KUKA KRL program: MyProgram_274().src

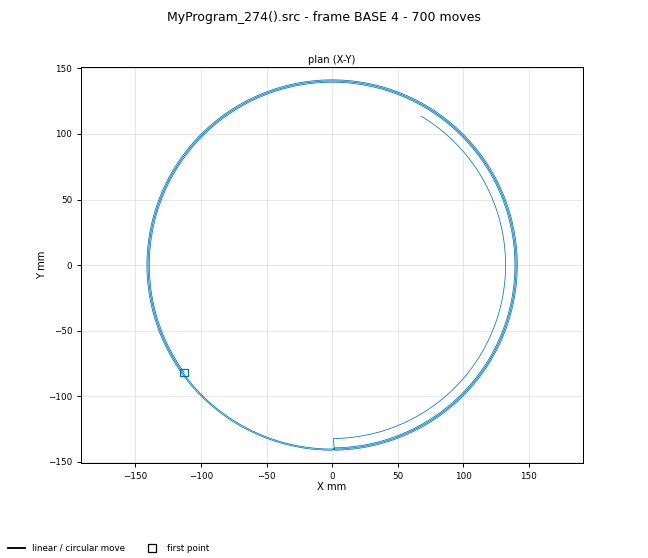
[picture p0: tool path of MyProgram_274().src in frame BASE 4, 700 of 700 moves have a stored position in this frame; points joined in program order, loops and branches not executed]
&ACCESS RVP
&REL 1
&PARAM TEMPLATE = C:\KRC\Roboter\Template\vorgabe
&PARAM EDITMASK = *
DEF MyProgram_274()
; ---- Setting reference (Base) ----
$BASE = BASE_DATA[4]

; --------------------------
; ---- Setting tool (TCP) ----
$TOOL = TOOL_DATA[3]
; --------------------------

$VEL.CP = VEL_APROX_PRINT
Startdeposition()
$VEL.CP = VEL_PRINT
LIN {X -112.8396,Y -81.9859,Z 171,A -142.2331,B 8.8363,C 0.3441,E1 8.7131,E2 233.8465} C_DIS
LIN {X -115.5145,Y -78.1719,Z 171,A -144.1484,B 8.8365,C 0.3397,E1 8.71,E2 235.7611} C_DIS
LIN {X -118.0573,Y -74.2762,Z 171,A -146.0937,B 8.8366,C 0.3357,E1 8.7071,E2 237.7098} C_DIS
LIN {X -120.4012,Y -70.4136,Z 171,A -147.8161,B 8.8369,C 0.3289,E1 8.7047,E2 239.4141} C_DIS
LIN {X -122.1598,Y -67.3164,Z 171,A -149.6524,B 8.8368,C 0.3315,E1 8.7021,E2 241.297} C_DIS
LIN {X -124.439,Y -62.9993,Z 171,A -151.4139,B 8.8371,C 0.3224,E1 8.6999,E2 243.0262} C_DIS
LIN {X -125.9748,Y -59.8691,Z 171,A -152.8774,B 8.8372,C 0.3192,E1 8.6981,E2 244.4928} C_DIS
LIN {X -127.4555,Y -56.6489,Z 171,A -154.3628,B 8.8374,C 0.3159,E1 8.6964,E2 245.981} C_DIS
LIN {X -128.9714,Y -53.1107,Z 171,A -156.2039,B 8.8374,C 0.3161,E1 8.6944,E2 247.854} C_DIS
LIN {X -130.384,Y -49.5416,Z 171,A -158.0959,B 8.8374,C 0.3171,E1 8.6925,E2 249.7847} C_DIS
LIN {X -131.9696,Y -45.1472,Z 171,A -159.478,B 8.8378,C 0.303,E1 8.6913,E2 251.0977} C_DIS
LIN {X -132.9491,Y -42.1728,Z 171,A -160.7834,B 8.8379,C 0.2998,E1 8.6901,E2 252.4044} C_DIS
LIN {X -133.9563,Y -38.8556,Z 171,A -162.2355,B 8.838,C 0.2964,E1 8.689,E2 253.8591} C_DIS
LIN {X -134.8227,Y -35.7326,Z 171,A -163.6103,B 8.8381,C 0.2934,E1 8.688,E2 255.2384} C_DIS
LIN {X -135.806,Y -31.8005,Z 171,A -165.4341,B 8.8382,C 0.2913,E1 8.6867,E2 257.081} C_DIS
LIN {X -136.6688,Y -27.8498,Z 171,A -167.0113,B 8.8384,C 0.2853,E1 8.6858,E2 258.6461} C_DIS
LIN {X -137.3745,Y -24.1335,Z 171,A -168.6614,B 8.8384,C 0.2824,E1 8.685,E2 260.3072} C_DIS
LIN {X -138.0563,Y -19.8611,Z 171,A -170.4155,B 8.8387,C 0.277,E1 8.6843,E2 262.0568} C_DIS
LIN {X -138.5691,Y -15.906,Z 171,A -172.5929,B 8.8385,C 0.281,E1 8.6836,E2 264.3005} C_DIS
LIN {X -139.0257,Y -11.2308,Z 171,A -173.9284,B 8.839,C 0.2658,E1 8.6833,E2 265.5598} C_DIS
LIN {X -139.2374,Y -8.1929,Z 171,A -175.9129,B 8.8387,C 0.2741,E1 8.6829,E2 267.6352} C_DIS
LIN {X -139.4478,Y -2.9637,Z 171,A -178.1689,B 8.8389,C 0.2696,E1 8.6828,E2 269.9025} C_DIS
LIN {X -139.4551,Y 2.5197,Z 171,A -179.7814,B 8.8394,C 0.2527,E1 8.6828,E2 271.4329} C_DIS
LIN {X -139.0897,Y 10.3992,Z 171,A 177.172,B 8.8397,C 0.2402,E1 8.6833,E2 274.4521} C_DIS
LIN {X -138.4769,Y 16.6784,Z 171,A 174.2904,B 8.8398,C 0.2375,E1 8.6841,E2 277.3677} C_DIS
LIN {X -137.9353,Y 20.6949,Z 171,A 172.3629,B 8.8398,C 0.2369,E1 8.6848,E2 279.3266} C_DIS
LIN {X -137.0859,Y 25.7227,Z 171,A 170.4087,B 8.84,C 0.2286,E1 8.6858,E2 281.2611} C_DIS
LIN {X -136.3153,Y 29.5315,Z 171,A 168.8667,B 8.8402,C 0.2232,E1 8.6867,E2 282.7947} C_DIS
LIN {X -135.543,Y 32.8954,Z 171,A 167.4503,B 8.8402,C 0.2192,E1 8.6876,E2 284.2094} C_DIS
LIN {X -134.7496,Y 36.0069,Z 171,A 166.0979,B 8.8403,C 0.216,E1 8.6885,E2 285.5647} C_DIS
LIN {X -133.815,Y 39.3382,Z 171,A 164.6154,B 8.8404,C 0.213,E1 8.6897,E2 287.0534} C_DIS
LIN {X -132.7678,Y 42.7402,Z 171,A 163.1696,B 8.8405,C 0.2087,E1 8.6909,E2 288.4957} C_DIS
LIN {X -131.6755,Y 45.9954,Z 171,A 161.7245,B 8.8405,C 0.2053,E1 8.6922,E2 289.9437} C_DIS
LIN {X -130.5628,Y 49.0642,Z 171,A 160.3436,B 8.8407,C 0.2023,E1 8.6935,E2 291.3282} C_DIS
LIN {X -129.2438,Y 52.4408,Z 171,A 158.8394,B 8.8407,C 0.1985,E1 8.6951,E2 292.8328} C_DIS
LIN {X -127.8789,Y 55.6868,Z 171,A 157.399,B 8.8408,C 0.1946,E1 8.6967,E2 294.2709} C_DIS
LIN {X -126.442,Y 58.8765,Z 171,A 155.9105,B 8.8409,C 0.1916,E1 8.6984,E2 295.7643} C_DIS
LIN {X -124.8829,Y 62.1157,Z 171,A 154.4187,B 8.8409,C 0.188,E1 8.7002,E2 297.2566} C_DIS
LIN {X -123.3331,Y 65.1378,Z 171,A 153.0073,B 8.8411,C 0.1846,E1 8.7021,E2 298.6685} C_DIS
LIN {X -121.1822,Y 69.0604,Z 171,A 150.9956,B 8.8411,C 0.1828,E1 8.7048,E2 300.7001} C_DIS
LIN {X -118.3623,Y 73.7886,Z 171,A 148.7116,B 8.8411,C 0.1775,E1 8.7081,E2 302.9845} C_DIS
LIN {X -116.2771,Y 77.034,Z 171,A 147.1234,B 8.8413,C 0.1737,E1 8.7106,E2 304.5716} C_DIS
LIN {X -113.7268,Y 80.7516,Z 171,A 145.2756,B 8.8413,C 0.1692,E1 8.7135,E2 306.417} C_DIS
LIN {X -111.0828,Y 84.3518,Z 171,A 143.2119,B 8.8413,C 0.1687,E1 8.717,E2 308.5072} C_DIS
LIN {X -109.099,Y 86.9014,Z 171,A 142.3013,B 8.8416,C 0.1587,E1 8.7185,E2 309.3647} C_DIS
LIN {X -107.0989,Y 89.3555,Z 171,A 140.6991,B 8.8416,C 0.1608,E1 8.7214,E2 311.0032} C_DIS
LIN {X -103.7086,Y 93.2685,Z 171,A 138.204,B 8.8415,C 0.1623,E1 8.7261,E2 313.5417} C_DIS
LIN {X -100.7826,Y 96.4226,Z 171,A 137.0283,B 8.8417,C 0.1486,E1 8.7282,E2 314.6424} C_DIS
LIN {X -98.5108,Y 98.7428,Z 171,A 134.866,B 8.8415,C 0.1598,E1 8.7327,E2 316.9059} C_DIS
LIN {X -94.6241,Y 102.4735,Z 171,A 132.7583,B 8.8416,C 0.1536,E1 8.737,E2 318.9986} C_DIS
LIN {X -91.1481,Y 105.5769,Z 171,A 131.3887,B 8.8419,C 0.1406,E1 8.7397,E2 320.299} C_DIS
LIN {X -88.0504,Y 108.1742,Z 171,A 129.1579,B 8.8417,C 0.1473,E1 8.7447,E2 322.5987} C_DIS
LIN {X -84.45,Y 111.0073,Z 171,A 127.7852,B 8.8419,C 0.1352,E1 8.7476,E2 323.9068} C_DIS
LIN {X -81.9039,Y 112.899,Z 171,A 126.4687,B 8.8419,C 0.1332,E1 8.7505,E2 325.2238} C_DIS
LIN {X -78.5911,Y 115.2304,Z 171,A 124.6683,B 8.8419,C 0.1327,E1 8.7547,E2 327.0397} C_DIS
LIN {X -73.9341,Y 118.2721,Z 171,A 122.4186,B 8.842,C 0.1285,E1 8.76,E2 329.283} C_DIS
LIN {X -67.4741,Y 122.0725,Z 171,A 119.5001,B 8.8421,C 0.1211,E1 8.767,E2 332.179} C_DIS
LIN {X -64.5541,Y 123.6396,Z 171,A 117.9816,B 8.8421,C 0.122,E1 8.7708,E2 333.7158} C_DIS
LIN {X -60.8845,Y 125.4897,Z 171,A 116.0518,B 8.8421,C 0.1241,E1 8.7757,E2 335.6743} C_DIS
LIN {X -56.6171,Y 127.4697,Z 171,A 114.3186,B 8.8421,C 0.1182,E1 8.78,E2 337.3812} C_DIS
LIN {X -51.3124,Y 129.6975,Z 171,A 112.0212,B 8.8422,C 0.1144,E1 8.7859,E2 339.6686} C_DIS
LIN {X -46.4257,Y 131.5259,Z 171,A 109.7822,B 8.8422,C 0.1139,E1 8.7918,E2 341.918} C_DIS
LIN {X -42.2053,Y 132.9387,Z 171,A 108.0067,B 8.8422,C 0.1113,E1 8.7965,E2 343.6856} C_DIS
LIN {X -39.0862,Y 133.8888,Z 171,A 106.6832,B 8.8422,C 0.1098,E1 8.8,E2 345.0061} C_DIS
LIN {X -35.8913,Y 134.7804,Z 171,A 105.2586,B 8.8422,C 0.1098,E1 8.8039,E2 346.4375} C_DIS
LIN {X -32.6408,Y 135.6043,Z 171,A 103.8694,B 8.8422,C 0.1091,E1 8.8077,E2 347.8272} C_DIS
LIN {X -28.9193,Y 136.4475,Z 171,A 101.9482,B 8.8422,C 0.1146,E1 8.813,E2 349.7913} C_DIS
LIN {X -25.2244,Y 137.1792,Z 171,A 99.9513,B 8.8422,C 0.1221,E1 8.8187,E2 351.8423} C_DIS
LIN {X -19.1774,Y 138.154,Z 171,A 98.2705,B 8.8423,C 0.1055,E1 8.823,E2 353.4189} C_DIS
LIN {X -15.6692,Y 138.5966,Z 171,A 96.225,B 8.8423,C 0.1161,E1 8.8289,E2 355.5369} C_DIS
LIN {X -10.9093,Y 139.0524,Z 171,A 94.6783,B 8.8423,C 0.1077,E1 8.8331,E2 357.0311} C_DIS
LIN {X -5.1132,Y 139.3843,Z 171,A 92.579,B 8.8423,C 0.1019,E1 8.8388,E2 359.0936} C_DIS
LIN {X -2.0688,Y 139.4626,Z 171,A 91.1654,B 8.8423,C 0.1049,E1 8.8428,E2 360.5269} C_DIS
LIN {X 1.9636,Y 139.4644,Z 171,A 89.1838,B 8.8423,C 0.1111,E1 8.8484,E2 362.548} C_DIS
LIN {X 5.4905,Y 139.3696,Z 171,A 87.8031,B 8.8423,C 0.1099,E1 8.8523,E2 363.9196} C_DIS
LIN {X 9.6693,Y 139.143,Z 171,A 86.2944,B 8.8423,C 0.1062,E1 8.8564,E2 365.4017} C_DIS
LIN {X 13.7603,Y 138.7979,Z 171,A 84.3806,B 8.8423,C 0.111,E1 8.8618,E2 367.343} C_DIS
LIN {X 17.0865,Y 138.4282,Z 171,A 83.2481,B 8.8423,C 0.1067,E1 8.8649,E2 368.4449} C_DIS
LIN {X 23.7404,Y 137.4444,Z 171,A 80.562,B 8.8423,C 0.1064,E1 8.8723,E2 371.1207} C_DIS
LIN {X 32.9569,Y 135.5281,Z 171,A 76.6599,B 8.8423,C 0.1094,E1 8.8829,E2 375.0263} C_DIS
LIN {X 36.1847,Y 134.7022,Z 171,A 75.3275,B 8.8423,C 0.1096,E1 8.8865,E2 376.3539} C_DIS
LIN {X 39.3671,Y 133.8066,Z 171,A 73.9683,B 8.8423,C 0.1107,E1 8.8901,E2 377.713} C_DIS
LIN {X 42.5681,Y 132.8228,Z 171,A 72.5899,B 8.8423,C 0.1119,E1 8.8938,E2 379.0915} C_DIS
LIN {X 46.0136,Y 131.6692,Z 171,A 71.1204,B 8.8423,C 0.1128,E1 8.8977,E2 380.558} C_DIS
LIN {X 49.2886,Y 130.4787,Z 171,A 69.7052,B 8.8423,C 0.1139,E1 8.9014,E2 381.971} C_DIS
LIN {X 52.7987,Y 129.0996,Z 171,A 67.8474,B 8.8421,C 0.1219,E1 8.9063,E2 383.8671} C_DIS
LIN {X 55.9083,Y 127.7831,Z 171,A 66.7646,B 8.8421,C 0.1172,E1 8.909,E2 384.9119} C_DIS
LIN {X 61.6274,Y 125.1238,Z 171,A 63.7194,B 8.8421,C 0.1297,E1 8.9168,E2 388.0136} C_DIS
LIN {X 65.6766,Y 123.0495,Z 171,A 62.2846,B 8.8421,C 0.1233,E1 8.9202,E2 389.3945} C_DIS
LIN {X 69.451,Y 120.9593,Z 171,A 60.5123,B 8.8421,C 0.1257,E1 8.9245,E2 391.1669} C_DIS
LIN {X 73.3803,Y 118.6167,Z 171,A 58.8119,B 8.8421,C 0.1248,E1 8.9285,E2 392.8451} C_DIS
LIN {X 75.557,Y 117.2423,Z 171,A 57.3892,B 8.842,C 0.1341,E1 8.932,E2 394.3136} C_DIS
LIN {X 78.2884,Y 115.4356,Z 171,A 55.6399,B 8.8418,C 0.1446,E1 8.9361,E2 396.1132} C_DIS
LIN {X 82.9019,Y 112.169,Z 171,A 54.0025,B 8.842,C 0.1342,E1 8.9396,E2 397.6659} C_DIS
LIN {X 86.2917,Y 109.5819,Z 171,A 52.2349,B 8.842,C 0.1376,E1 8.9435,E2 399.4358} C_DIS
LIN {X 89.8009,Y 106.7252,Z 171,A 50.3797,B 8.8419,C 0.1409,E1 8.9475,E2 401.2909} C_DIS
LIN {X 93.2101,Y 103.761,Z 171,A 48.3871,B 8.8417,C 0.1473,E1 8.9517,E2 403.3013} C_DIS
LIN {X 96.2147,Y 100.9812,Z 171,A 46.8805,B 8.8417,C 0.1469,E1 8.9548,E2 404.7864} C_DIS
LIN {X 99.2554,Y 97.9949,Z 171,A 45.119,B 8.8417,C 0.1507,E1 8.9582,E2 406.5499} C_DIS
LIN {X 104.0961,Y 92.8361,Z 171,A 42.2829,B 8.8417,C 0.1553,E1 8.9636,E2 409.3782} C_DIS
LIN {X 107.0425,Y 89.4227,Z 171,A 40.4474,B 8.8415,C 0.159,E1 8.9669,E2 411.2124} C_DIS
LIN {X 109.9181,Y 85.8638,Z 171,A 38.6101,B 8.8415,C 0.1623,E1 8.9701,E2 413.0452} C_DIS
LIN {X 112.6381,Y 82.2633,Z 171,A 36.7415,B 8.8415,C 0.1669,E1 8.9732,E2 414.9166} C_DIS
LIN {X 115.3005,Y 78.488,Z 171,A 34.8656,B 8.8413,C 0.1709,E1 8.9762,E2 416.7906} C_DIS
LIN {X 117.4671,Y 75.2058,Z 171,A 33.1544,B 8.8413,C 0.1769,E1 8.9788,E2 418.5148} C_DIS
LIN {X 120.6812,Y 69.932,Z 171,A 30.8465,B 8.8412,C 0.1781,E1 8.9821,E2 420.7952} C_DIS
LIN {X 122.717,Y 66.2955,Z 171,A 29.0961,B 8.8411,C 0.1833,E1 8.9845,E2 422.5514} C_DIS
LIN {X 124.4992,Y 62.8809,Z 171,A 27.6221,B 8.8411,C 0.1849,E1 8.9863,E2 424.0126} C_DIS
LIN {X 126.3601,Y 59.0537,Z 171,A 26.0265,B 8.8411,C 0.186,E1 8.9882,E2 425.5901} C_DIS
LIN {X 129.537,Y 51.7135,Z 171,A 22.7043,B 8.8408,C 0.1956,E1 8.9919,E2 428.9191} C_DIS
LIN {X 130.6783,Y 48.7557,Z 171,A 21.3935,B 8.8408,C 0.1993,E1 8.9932,E2 430.2319} C_DIS
LIN {X 131.9118,Y 45.3138,Z 171,A 19.9147,B 8.8407,C 0.2028,E1 8.9945,E2 431.7089} C_DIS
LIN {X 132.9524,Y 42.1625,Z 171,A 18.5801,B 8.8406,C 0.2059,E1 8.9957,E2 433.0408} C_DIS
LIN {X 133.9281,Y 38.9519,Z 171,A 17.2266,B 8.8406,C 0.2092,E1 8.9968,E2 434.3922} C_DIS
LIN {X 134.8223,Y 35.7344,Z 171,A 15.8718,B 8.8404,C 0.2126,E1 8.9978,E2 435.7459} C_DIS
LIN {X 135.7933,Y 31.8549,Z 171,A 13.7509,B 8.84,C 0.228,E1 8.9992,E2 437.9288} C_DIS
LIN {X 136.7354,Y 27.5224,Z 171,A 12.4936,B 8.8402,C 0.2204,E1 8.9999,E2 439.116} C_DIS
LIN {X 137.2961,Y 24.5712,Z 171,A 10.5895,B 8.8398,C 0.2391,E1 9.0008,E2 441.1061} C_DIS
LIN {X 138.1564,Y 19.161,Z 171,A 9.0747,B 8.84,C 0.2289,E1 9.0014,E2 442.5296} C_DIS
LIN {X 138.8069,Y 13.666,Z 171,A 6.988,B 8.84,C 0.2312,E1 9.0021,E2 444.5945} C_DIS
LIN {X 139.0649,Y 10.7379,Z 171,A 5.5151,B 8.8397,C 0.2407,E1 9.0024,E2 446.1024} C_DIS
LIN {X 139.3175,Y 6.6909,Z 171,A 3.7156,B 8.8395,C 0.2486,E1 9.0027,E2 447.9204} C_DIS
LIN {X 139.482,Y -0.0033,Z 171,A 1.0113,B 8.8393,C 0.2555,E1 9.0027,E2 450.6215} C_DIS
LIN {X 139.398,Y -4.764,Z 171,A -1.0684,B 8.8391,C 0.264,E1 9.0026,E2 452.7187} C_DIS
LIN {X 139.2074,Y -8.6797,Z 171,A -2.2767,B 8.8391,C 0.2596,E1 9.0024,E2 453.8771} C_DIS
LIN {X 138.7329,Y -14.4036,Z 171,A -4.4383,B 8.8391,C 0.2619,E1 9.0019,E2 456.0157} C_DIS
LIN {X 138.2511,Y -18.4595,Z 171,A -6.2004,B 8.8389,C 0.2687,E1 9.0013,E2 457.7903} C_DIS
LIN {X 137.7385,Y -21.9657,Z 171,A -7.7867,B 8.8387,C 0.2758,E1 9.0006,E2 459.3948} C_DIS
LIN {X 137.1068,Y -25.6126,Z 171,A -9.5205,B 8.8384,C 0.285,E1 8.9997,E2 461.1574} C_DIS
LIN {X 136.3613,Y -29.3186,Z 171,A -10.3994,B 8.8387,C 0.2741,E1 8.9993,E2 461.9514} C_DIS
LIN {X 134.8966,Y -35.4555,Z 171,A -13.0858,B 8.8385,C 0.2837,E1 8.9975,E2 464.6527} C_DIS
LIN {X 133.7501,Y -39.5598,Z 171,A -14.9247,B 8.8382,C 0.2906,E1 8.9961,E2 466.5048} C_DIS
LIN {X 132.7916,Y -42.6657,Z 171,A -16.2571,B 8.8382,C 0.2943,E1 8.9949,E2 467.8381} C_DIS
LIN {X 131.6179,Y -46.1617,Z 171,A -17.7427,B 8.838,C 0.2978,E1 8.9936,E2 469.3216} C_DIS
LIN {X 129.7219,Y -51.2517,Z 171,A -19.9243,B 8.8378,C 0.3028,E1 8.9915,E2 471.4991} C_DIS
LIN {X 128.6777,Y -53.8139,Z 171,A -21.0297,B 8.8378,C 0.3052,E1 8.9903,E2 472.6017} C_DIS
LIN {X 125.5512,Y -60.7557,Z 171,A -23.9014,B 8.8376,C 0.3078,E1 8.987,E2 475.4437} C_DIS
LIN {X 123.9373,Y -63.9846,Z 171,A -25.5965,B 8.8373,C 0.3165,E1 8.9848,E2 477.1679} C_DIS
LIN {X 121.4883,Y -68.5207,Z 171,A -27.7719,B 8.8371,C 0.3233,E1 8.9819,E2 479.3529} C_DIS
LIN {X 119.1489,Y -72.513,Z 171,A -29.8109,B 8.8368,C 0.3313,E1 8.9789,E2 481.4117} C_DIS
LIN {X 116.1482,Y -77.2275,Z 171,A -31.9345,B 8.8368,C 0.3331,E1 8.9757,E2 483.5155} C_DIS
LIN {X 112.7181,Y -82.1535,Z 171,A -34.1008,B 8.8368,C 0.3324,E1 8.9723,E2 485.6457} C_DIS
LIN {X 108.5305,Y -87.6104,Z 171,A -37.0675,B 8.8364,C 0.3422,E1 8.9672,E2 488.6336} C_DIS
LIN {X 105.9236,Y -90.7456,Z 171,A -38.816,B 8.8362,C 0.3477,E1 8.964,E2 490.3934} C_DIS
LIN {X 102.2707,Y -94.8428,Z 171,A -41.2535,B 8.8358,C 0.3567,E1 8.9594,E2 492.8566} C_DIS
LIN {X 99.7954,Y -97.4444,Z 171,A -42.5038,B 8.8358,C 0.355,E1 8.957,E2 494.0795} C_DIS
LIN {X 96.4987,Y -100.7098,Z 171,A -44.3704,B 8.8358,C 0.3581,E1 8.9533,E2 495.9428} C_DIS
LIN {X 92.2815,Y -104.5877,Z 171,A -46.9905,B 8.8353,C 0.3687,E1 8.9478,E2 498.5996} C_DIS
LIN {X 89.2531,Y -107.1842,Z 171,A -48.3219,B 8.8355,C 0.3652,E1 8.945,E2 499.8929} C_DIS
LIN {X 85.6888,Y -110.0543,Z 171,A -50.1537,B 8.8354,C 0.3677,E1 8.941,E2 501.7203} C_DIS
LIN {X 82.0331,Y -112.8054,Z 171,A -51.9295,B 8.8354,C 0.3688,E1 8.9371,E2 503.4844} C_DIS
LIN {X 77.9243,Y -115.6821,Z 171,A -53.9797,B 8.8352,C 0.3722,E1 8.9323,E2 505.5352} C_DIS
LIN {X 73.1326,Y -118.7684,Z 171,A -56.5354,B 8.8348,C 0.3807,E1 8.9262,E2 508.1208} C_DIS
LIN {X 69.1462,Y -121.1332,Z 171,A -58.0542,B 8.8351,C 0.3754,E1 8.9227,E2 509.5913} C_DIS
LIN {X 66.3121,Y -122.708,Z 171,A -59.6043,B 8.8348,C 0.3821,E1 8.9188,E2 511.1709} C_DIS
LIN {X 62.9686,Y -124.4546,Z 171,A -61.0442,B 8.8348,C 0.3819,E1 8.9153,E2 512.5978} C_DIS
LIN {X 59.6859,Y -126.0623,Z 171,A -62.6688,B 8.8346,C 0.3866,E1 8.9111,E2 514.2396} C_DIS
LIN {X 53.7609,Y -128.6999,Z 171,A -64.8604,B 8.8349,C 0.38,E1 8.9057,E2 516.372} C_DIS
LIN {X 49.776,Y -130.2955,Z 171,A -67.0581,B 8.8344,C 0.3912,E1 8.8998,E2 518.6276} C_DIS
LIN {X 42.2179,Y -132.9347,Z 171,A -70.1748,B 8.8344,C 0.3911,E1 8.8917,E2 521.7245} C_DIS
LIN {X 38.9371,Y -133.9325,Z 171,A -71.5708,B 8.8344,C 0.3921,E1 8.8879,E2 523.1199} C_DIS
LIN {X 35.5501,Y -134.8714,Z 171,A -73.8381,B 8.8335,C 0.4104,E1 8.8815,E2 525.4944} C_DIS
LIN {X 29.5341,Y -136.3147,Z 171,A -76.3675,B 8.8335,C 0.412,E1 8.8746,E2 528.0238} C_DIS
LIN {X 23.4129,Y -137.4992,Z 171,A -78.2991,B 8.8339,C 0.4008,E1 8.8695,E2 529.8761} C_DIS
LIN {X 17.17,Y -138.4183,Z 171,A -80.6166,B 8.8341,C 0.3966,E1 8.8632,E2 532.1597} C_DIS
LIN {X 14.6108,Y -138.7106,Z 171,A -81.7114,B 8.8341,C 0.3978,E1 8.8601,E2 533.2598} C_DIS
LIN {X 10.9284,Y -139.0508,Z 171,A -83.4594,B 8.8339,C 0.403,E1 8.8552,E2 535.0383} C_DIS
LIN {X 6.5695,Y -139.3236,Z 171,A -85.1821,B 8.8339,C 0.402,E1 8.8504,E2 536.7527} C_DIS
LIN {X 2.1826,Y -139.4608,Z 171,A -86.8306,B 8.834,C 0.3993,E1 8.8459,E2 538.382} C_DIS
LIN {X 2.1826,Y -139.4608,Z 171,A -86.8306,B 8.834,C 0.3993,E1 8.8459,E2 538.382} C_DIS
Enddeposition()
LIN {X 1.0238,Y -140.3815,Z 171,A -86.8855,B 8.834,C 0.3961,E1 8.8457,E2 538.416} C_DIS
Startdeposition()
$VEL.CP = VEL_PRINT
LIN {X 4.1318,Y -140.3274,Z 171,A -85.3306,B 8.8343,C 0.39,E1 8.8501,E2 536.8229} C_DIS
LIN {X 8.0102,Y -140.1607,Z 171,A -83.7344,B 8.8343,C 0.3893,E1 8.8546,E2 535.2242} C_DIS
LIN {X 12.2354,Y -139.8544,Z 171,A -82.0924,B 8.8343,C 0.3905,E1 8.8591,E2 533.5928} C_DIS
LIN {X 16.2117,Y -139.4494,Z 171,A -80.5317,B 8.8343,C 0.3913,E1 8.8634,E2 532.0405} C_DIS
LIN {X 19.4391,Y -139.0362,Z 171,A -78.7545,B 8.8347,C 0.3812,E1 8.8685,E2 530.2028} C_DIS
LIN {X 23.3049,Y -138.4401,Z 171,A -77.5282,B 8.8344,C 0.388,E1 8.8718,E2 529.0248} C_DIS
LIN {X 27.682,Y -137.6319,Z 171,A -75.7455,B 8.8344,C 0.3875,E1 8.8766,E2 527.2454} C_DIS
LIN {X 31.0665,Y -136.9074,Z 171,A -74.326,B 8.8344,C 0.3863,E1 8.8805,E2 525.824} C_DIS
LIN {X 36.623,Y -135.5274,Z 171,A -72.0018,B 8.8346,C 0.3846,E1 8.8868,E2 523.4999} C_DIS
LIN {X 40.8332,Y -134.3183,Z 171,A -70.2501,B 8.8346,C 0.3837,E1 8.8915,E2 521.7517} C_DIS
LIN {X 45.0838,Y -132.9539,Z 171,A -68.3699,B 8.8347,C 0.3806,E1 8.8965,E2 519.8625} C_DIS
LIN {X 48.9238,Y -131.5874,Z 171,A -66.9169,B 8.8347,C 0.3833,E1 8.9002,E2 518.436} C_DIS
LIN {X 52.0122,Y -130.3981,Z 171,A -65.4085,B 8.8348,C 0.3783,E1 8.9042,E2 516.9057} C_DIS
LIN {X 60.0934,Y -126.8766,Z 171,A -61.6465,B 8.8352,C 0.3702,E1 8.9139,E2 513.1192} C_DIS
LIN {X 64.7345,Y -124.573,Z 171,A -59.6916,B 8.8352,C 0.3706,E1 8.9187,E2 511.1837} C_DIS
LIN {X 68.817,Y -122.366,Z 171,A -57.4249,B 8.8356,C 0.3596,E1 8.9243,E2 508.8658} C_DIS
LIN {X 72.5549,Y -120.1874,Z 171,A -55.7857,B 8.8356,C 0.3596,E1 8.9282,E2 507.2419} C_DIS
LIN {X 75.6984,Y -118.2327,Z 171,A -54.5623,B 8.8354,C 0.3634,E1 8.931,E2 506.0553} C_DIS
LIN {X 80.7722,Y -114.8264,Z 171,A -52.0681,B 8.8356,C 0.3591,E1 8.9368,E2 503.5589} C_DIS
LIN {X 84.3683,Y -112.2108,Z 171,A -50.2804,B 8.8357,C 0.3564,E1 8.9408,E2 501.7731} C_DIS
LIN {X 87.8737,Y -109.4876,Z 171,A -48.4632,B 8.8359,C 0.3529,E1 8.9448,E2 499.9534} C_DIS
LIN {X 90.6988,Y -107.1589,Z 171,A -47.0712,B 8.8359,C 0.3522,E1 8.9477,E2 498.5735} C_DIS
LIN {X 93.7356,Y -104.5125,Z 171,A -45.4316,B 8.836,C 0.349,E1 8.9512,E2 496.9329} C_DIS
LIN {X 96.7611,Y -101.7182,Z 171,A -43.7169,B 8.8362,C 0.3448,E1 8.9547,E2 495.212} C_DIS
LIN {X 99.7705,Y -98.768,Z 171,A -42.1265,B 8.8362,C 0.3441,E1 8.9578,E2 493.6371} C_DIS
LIN {X 102.1697,Y -96.2837,Z 171,A -40.5725,B 8.8365,C 0.3377,E1 8.9608,E2 492.0625} C_DIS
LIN {X 105.3051,Y -92.8443,Z 171,A -38.7786,B 8.8365,C 0.3359,E1 8.9641,E2 490.2807} C_DIS
LIN {X 108.2666,Y -89.3733,Z 171,A -36.9731,B 8.8366,C 0.3329,E1 8.9674,E2 488.4807} C_DIS
LIN {X 111.3984,Y -85.4376,Z 171,A -34.7026,B 8.837,C 0.3231,E1 8.9713,E2 486.1794} C_DIS
LIN {X 113.4331,Y -82.7182,Z 171,A -33.0274,B 8.8374,C 0.3131,E1 8.9741,E2 484.4643} C_DIS
LIN {X 116.3317,Y -78.5886,Z 171,A -31.5719,B 8.837,C 0.322,E1 8.9763,E2 483.0867} C_DIS
LIN {X 119.4389,Y -73.7816,Z 171,A -29.1586,B 8.8373,C 0.3143,E1 8.9799,E2 480.6609} C_DIS
LIN {X 121.7033,Y -69.9834,Z 171,A -27.4019,B 8.8374,C 0.3108,E1 8.9824,E2 478.9086} C_DIS
LIN {X 123.8744,Y -66.0646,Z 171,A -25.1968,B 8.8379,C 0.2974,E1 8.9854,E2 476.6518} C_DIS
LIN {X 125.8978,Y -62.1159,Z 171,A -23.9295,B 8.8376,C 0.3052,E1 8.9869,E2 475.4544} C_DIS
LIN {X 127.8212,Y -58.0607,Z 171,A -21.9896,B 8.8379,C 0.2978,E1 8.9892,E2 473.4985} C_DIS
LIN {X 129.4743,Y -54.2687,Z 171,A -20.4252,B 8.8379,C 0.2961,E1 8.9909,E2 471.9485} C_DIS
LIN {X 130.7574,Y -51.1001,Z 171,A -19.0643,B 8.838,C 0.293,E1 8.9923,E2 470.5906} C_DIS
LIN {X 132.3306,Y -46.8818,Z 171,A -17.1373,B 8.8383,C 0.2859,E1 8.9941,E2 468.6501} C_DIS
LIN {X 133.6429,Y -42.9924,Z 171,A -15.6481,B 8.8383,C 0.2855,E1 8.9954,E2 467.1836} C_DIS
LIN {X 135.4417,Y -36.9443,Z 171,A -13.1144,B 8.8385,C 0.2793,E1 8.9974,E2 464.6527} C_DIS
LIN {X 137.0278,Y -30.5396,Z 171,A -10.4879,B 8.8387,C 0.2732,E1 8.9991,E2 462.0323} C_DIS
LIN {X 137.8928,Y -26.35,Z 171,A -8.7577,B 8.8388,C 0.2686,E1 9,E2 460.3024} C_DIS
LIN {X 138.5087,Y -22.8939,Z 171,A -7.2867,B 8.839,C 0.2635,E1 9.0007,E2 458.825} C_DIS
LIN {X 139.0948,Y -19.0256,Z 171,A -5.666,B 8.8391,C 0.2584,E1 9.0014,E2 457.1997} C_DIS
LIN {X 139.4974,Y -15.8067,Z 171,A -4.3185,B 8.8392,C 0.254,E1 9.0018,E2 455.8478} C_DIS
LIN {X 139.9688,Y -10.8596,Z 171,A -2.3558,B 8.8394,C 0.2497,E1 9.0023,E2 453.8917} C_DIS
LIN {X 140.2403,Y -6.4659,Z 171,A -0.6391,B 8.8394,C 0.2463,E1 9.0025,E2 452.1838} C_DIS
LIN {X 140.3671,Y -2.4266,Z 171,A 0.9547,B 8.8396,C 0.2428,E1 9.0027,E2 450.5955} C_DIS
LIN {X 140.3821,Y 1.478,Z 171,A 2.4807,B 8.8396,C 0.2397,E1 9.0027,E2 449.0769} C_DIS
LIN {X 140.3152,Y 4.5708,Z 171,A 3.8494,B 8.8398,C 0.2336,E1 9.0025,E2 447.6932} C_DIS
LIN {X 140.1221,Y 8.6367,Z 171,A 5.384,B 8.8398,C 0.2317,E1 9.0023,E2 446.1736} C_DIS
LIN {X 139.8247,Y 12.5865,Z 171,A 7.0696,B 8.84,C 0.2255,E1 9.0019,E2 444.4776} C_DIS
LIN {X 139.3433,Y 17.1011,Z 171,A 8.8608,B 8.8401,C 0.2216,E1 9.0013,E2 442.6928} C_DIS
LIN {X 138.3871,Y 23.623,Z 171,A 11.5422,B 8.8403,C 0.2141,E1 9.0002,E2 440.0104} C_DIS
LIN {X 137.6437,Y 27.624,Z 171,A 13.1159,B 8.8403,C 0.2114,E1 8.9994,E2 438.4467} C_DIS
LIN {X 136.3576,Y 33.4006,Z 171,A 15.508,B 8.8405,C 0.2051,E1 8.9979,E2 436.0557} C_DIS
LIN {X 135.3013,Y 37.4486,Z 171,A 17.1516,B 8.8405,C 0.2018,E1 8.9967,E2 434.419} C_DIS
LIN {X 134.3714,Y 40.6597,Z 171,A 18.3622,B 8.8405,C 0.2016,E1 8.9957,E2 433.2274} C_DIS
LIN {X 133.3303,Y 43.9534,Z 171,A 19.8832,B 8.8407,C 0.1952,E1 8.9944,E2 431.6909} C_DIS
LIN {X 132.2622,Y 47.0715,Z 171,A 21.2301,B 8.8408,C 0.1915,E1 8.9932,E2 430.3428} C_DIS
LIN {X 130.8734,Y 50.8018,Z 171,A 22.7104,B 8.8408,C 0.1904,E1 8.9917,E2 428.88} C_DIS
LIN {X 128.7332,Y 56.0047,Z 171,A 25.1032,B 8.841,C 0.1821,E1 8.9891,E2 426.4732} C_DIS
LIN {X 127.2605,Y 59.2754,Z 171,A 26.6422,B 8.8411,C 0.1765,E1 8.9873,E2 424.9235} C_DIS
LIN {X 125.2902,Y 63.3337,Z 171,A 28.3379,B 8.8411,C 0.1751,E1 8.9852,E2 423.2455} C_DIS
LIN {X 123.4837,Y 66.7918,Z 171,A 30.0087,B 8.8413,C 0.1693,E1 8.983,E2 421.5637} C_DIS
LIN {X 121.5973,Y 70.1666,Z 171,A 32.1022,B 8.8415,C 0.1537,E1 8.98,E2 419.4023} C_DIS
LIN {X 118.7758,Y 74.8434,Z 171,A 33.7112,B 8.8414,C 0.1623,E1 8.9778,E2 417.8726} C_DIS
LIN {X 116.0679,Y 78.9782,Z 171,A 35.729,B 8.8414,C 0.1574,E1 8.9746,E2 415.8537} C_DIS
LIN {X 113.4439,Y 82.7033,Z 171,A 37.5722,B 8.8415,C 0.1535,E1 8.9716,E2 414.0118} C_DIS
LIN {X 110.6612,Y 86.3914,Z 171,A 39.4319,B 8.8416,C 0.1498,E1 8.9685,E2 412.1546} C_DIS
LIN {X 107.7905,Y 89.9475,Z 171,A 41.2836,B 8.8416,C 0.1459,E1 8.9652,E2 410.3038} C_DIS
LIN {X 105.1313,Y 93.041,Z 171,A 42.9523,B 8.8417,C 0.1422,E1 8.9621,E2 408.6339} C_DIS
LIN {X 101.8972,Y 96.5727,Z 171,A 44.8089,B 8.8417,C 0.1403,E1 8.9586,E2 406.7893} C_DIS
LIN {X 98.743,Y 99.7953,Z 171,A 46.6153,B 8.8418,C 0.1373,E1 8.9551,E2 404.9867} C_DIS
LIN {X 95.6782,Y 102.737,Z 171,A 48.3526,B 8.8418,C 0.1338,E1 8.9515,E2 403.2484} C_DIS
LIN {X 92.1876,Y 105.8805,Z 171,A 50.2447,B 8.8419,C 0.1307,E1 8.9476,E2 401.3589} C_DIS
LIN {X 88.6535,Y 108.8569,Z 171,A 52.1187,B 8.8419,C 0.1275,E1 8.9435,E2 399.486} C_DIS
LIN {X 85.0556,Y 111.6908,Z 171,A 53.91,B 8.8419,C 0.1259,E1 8.9396,E2 397.7043} C_DIS
LIN {X 78.4965,Y 116.394,Z 171,A 57.2296,B 8.8421,C 0.12,E1 8.932,E2 394.381} C_DIS
LIN {X 74.708,Y 118.8613,Z 171,A 59.1427,B 8.8421,C 0.1157,E1 8.9275,E2 392.4591} C_DIS
LIN {X 70.5916,Y 121.3512,Z 171,A 61.0485,B 8.8421,C 0.1141,E1 8.9229,E2 390.5605} C_DIS
LIN {X 66.472,Y 123.6555,Z 171,A 63.4785,B 8.8423,C 0.1007,E1 8.9168,E2 388.0657} C_DIS
LIN {X 61.8286,Y 126.0396,Z 171,A 65.0025,B 8.8422,C 0.1109,E1 8.9132,E2 386.6195} C_DIS
LIN {X 57.6567,Y 128.002,Z 171,A 66.8195,B 8.8422,C 0.11,E1 8.9086,E2 384.8108} C_DIS
LIN {X 53.3448,Y 129.8602,Z 171,A 68.8542,B 8.8422,C 0.1054,E1 8.9033,E2 382.7613} C_DIS
LIN {X 49.5298,Y 131.3605,Z 171,A 70.3918,B 8.8422,C 0.1065,E1 8.8994,E2 381.2409} C_DIS
LIN {X 46.2643,Y 132.5458,Z 171,A 71.8779,B 8.8422,C 0.1037,E1 8.8954,E2 379.7463} C_DIS
LIN {X 42.5851,Y 133.773,Z 171,A 73.3383,B 8.8422,C 0.1049,E1 8.8916,E2 378.3017} C_DIS
LIN {X 39.649,Y 134.6726,Z 171,A 74.6267,B 8.8422,C 0.1031,E1 8.8882,E2 377.0091} C_DIS
LIN {X 35.8453,Y 135.7348,Z 171,A 76.8062,B 8.8424,C 0.0903,E1 8.8821,E2 374.7574} C_DIS
LIN {X 31.0409,Y 136.9133,Z 171,A 78.2764,B 8.8423,C 0.1003,E1 8.8783,E2 373.3579} C_DIS
LIN {X 26.6467,Y 137.836,Z 171,A 80.077,B 8.8423,C 0.0999,E1 8.8734,E2 371.5618} C_DIS
LIN {X 23.3572,Y 138.4314,Z 171,A 81.5533,B 8.8423,C 0.097,E1 8.8693,E2 370.0717} C_DIS
LIN {X 19.0358,Y 139.0936,Z 171,A 83.256,B 8.8423,C 0.0979,E1 8.8646,E2 368.3799} C_DIS
LIN {X 14.806,Y 139.6052,Z 171,A 84.9546,B 8.8423,C 0.0982,E1 8.8599,E2 366.687} C_DIS
LIN {X 10.9557,Y 139.9618,Z 171,A 86.6116,B 8.8423,C 0.0963,E1 8.8552,E2 365.0206} C_DIS
LIN {X 6.6064,Y 140.2332,Z 171,A 88.3467,B 8.8423,C 0.0969,E1 8.8504,E2 363.2918} C_DIS
LIN {X 3.0996,Y 140.3559,Z 171,A 89.8526,B 8.8423,C 0.0954,E1 8.8462,E2 361.7772} C_DIS
LIN {X -1.1349,Y 140.384,Z 171,A 91.4408,B 8.8423,C 0.0981,E1 8.8418,E2 360.2075} C_DIS
LIN {X -4.9504,Y 140.3017,Z 171,A 93.1444,B 8.8423,C 0.0955,E1 8.837,E2 358.4861} C_DIS
LIN {X -9.3577,Y 140.0772,Z 171,A 94.7672,B 8.8423,C 0.0992,E1 8.8325,E2 356.8868} C_DIS
LIN {X -12.77,Y 139.8075,Z 171,A 96.2601,B 8.8423,C 0.0978,E1 8.8284,E2 355.3825} C_DIS
LIN {X -16.5121,Y 139.4135,Z 171,A 97.7787,B 8.8423,C 0.0986,E1 8.8241,E2 353.8669} C_DIS
LIN {X -19.5662,Y 139.018,Z 171,A 99.2922,B 8.8423,C 0.0942,E1 8.8199,E2 352.3215} C_DIS
LIN {X -22.8,Y 138.5244,Z 171,A 100.6119,B 8.8423,C 0.0952,E1 8.8162,E2 351.0045} C_DIS
LIN {X -29.4133,Y 137.2721,Z 171,A 103.1967,B 8.8423,C 0.0999,E1 8.8092,E2 348.4421} C_DIS
LIN {X -33.7945,Y 136.2616,Z 171,A 105.0563,B 8.8423,C 0.1007,E1 8.8042,E2 346.5807} C_DIS
LIN {X -37.4953,Y 135.2883,Z 171,A 106.4611,B 8.8423,C 0.1048,E1 8.8004,E2 345.1968} C_DIS
LIN {X -40.4002,Y 134.4509,Z 171,A 107.7058,B 8.8423,C 0.1057,E1 8.7971,E2 343.9516} C_DIS
LIN {X -44.0837,Y 133.2869,Z 171,A 109.1321,B 8.8422,C 0.1099,E1 8.7934,E2 342.5454} C_DIS
LIN {X -49.9578,Y 131.2001,Z 171,A 111.9788,B 8.8422,C 0.1069,E1 8.7858,E2 339.6625} C_DIS
LIN {X -53.7982,Y 129.6708,Z 171,A 113.6212,B 8.8422,C 0.1096,E1 8.7816,E2 338.027} C_DIS
LIN {X -56.9835,Y 128.3031,Z 171,A 115.4238,B 8.8422,C 0.1042,E1 8.7768,E2 336.1762} C_DIS
LIN {X -60.504,Y 126.6804,Z 171,A 116.6428,B 8.8422,C 0.1128,E1 8.7739,E2 335.0047} C_DIS
LIN {X -63.4392,Y 125.2365,Z 171,A 117.9717,B 8.8422,C 0.1147,E1 8.7706,E2 333.6777} C_DIS
LIN {X -66.7186,Y 123.523,Z 171,A 119.4522,B 8.8421,C 0.1173,E1 8.7669,E2 332.2023} C_DIS
LIN {X -70.6893,Y 121.2947,Z 171,A 121.4451,B 8.8421,C 0.1176,E1 8.7621,E2 330.1939} C_DIS
LIN {X -74.5136,Y 118.9836,Z 171,A 123.2157,B 8.8421,C 0.1214,E1 8.7579,E2 328.4316} C_DIS
LIN {X -78.0855,Y 116.67,Z 171,A 125.0413,B 8.8421,C 0.1226,E1 8.7536,E2 326.5963} C_DIS
LIN {X -81.6345,Y 114.2148,Z 171,A 127.1353,B 8.8421,C 0.1197,E1 8.7487,E2 324.4615} C_DIS
LIN {X -84.8157,Y 111.8731,Z 171,A 128.899,B 8.8421,C 0.1198,E1 8.7448,E2 322.68} C_DIS
LIN {X -88.4973,Y 108.9843,Z 171,A 130.4323,B 8.8419,C 0.13,E1 8.7415,E2 321.1965} C_DIS
LIN {X -95.4254,Y 102.9724,Z 171,A 135.0458,B 8.842,C 0.122,E1 8.7317,E2 316.4753} C_DIS
LIN {X -100.4436,Y 98.0836,Z 171,A 136.7753,B 8.8416,C 0.1477,E1 8.7286,E2 314.8931} C_DIS
LIN {X -105.2461,Y 92.9111,Z 171,A 140.4563,B 8.8418,C 0.1401,E1 8.7215,E2 311.1131} C_DIS
LIN {X -108.3917,Y 89.2223,Z 171,A 141.9721,B 8.8416,C 0.1526,E1 8.7189,E2 309.6584} C_DIS
LIN {X -111.1594,Y 85.7491,Z 171,A 143.7967,B 8.8415,C 0.1566,E1 8.7158,E2 307.8342} C_DIS
LIN {X -113.7781,Y 82.2423,Z 171,A 145.582,B 8.8415,C 0.1608,E1 8.7128,E2 306.0507} C_DIS
LIN {X -116.2015,Y 78.7809,Z 171,A 147.3963,B 8.8414,C 0.1634,E1 8.7099,E2 304.2268} C_DIS
LIN {X -120.8168,Y 71.5032,Z 171,A 150.7059,B 8.8411,C 0.1757,E1 8.7051,E2 300.9473} C_DIS
LIN {X -122.5276,Y 68.5295,Z 171,A 152.3207,B 8.8411,C 0.1757,E1 8.7028,E2 299.3067} C_DIS
LIN {X -124.6025,Y 64.6784,Z 171,A 154.2152,B 8.8411,C 0.1784,E1 8.7003,E2 297.4001} C_DIS
LIN {X -126.4228,Y 61.0431,Z 171,A 155.7825,B 8.841,C 0.1843,E1 8.6984,E2 295.8463} C_DIS
LIN {X -128.1823,Y 57.2534,Z 171,A 157.4489,B 8.8408,C 0.1895,E1 8.6965,E2 294.1865} C_DIS
LIN {X -129.4148,Y 54.4112,Z 171,A 158.817,B 8.8408,C 0.1911,E1 8.695,E2 292.8065} C_DIS
LIN {X -130.7371,Y 51.1524,Z 171,A 160.1999,B 8.8408,C 0.1959,E1 8.6935,E2 291.4318} C_DIS
LIN {X -131.7968,Y 48.3624,Z 171,A 161.6227,B 8.8408,C 0.1959,E1 8.6921,E2 289.9841} C_DIS
LIN {X -132.9974,Y 44.9531,Z 171,A 163.0581,B 8.8406,C 0.2005,E1 8.6908,E2 288.5553} C_DIS
LIN {X -134.2305,Y 41.1201,Z 171,A 164.6236,B 8.8405,C 0.2064,E1 8.6895,E2 287.0014} C_DIS
LIN {X -135.2243,Y 37.724,Z 171,A 166.1067,B 8.8404,C 0.2098,E1 8.6884,E2 285.5148} C_DIS
LIN {X -136.0717,Y 34.5428,Z 171,A 167.5076,B 8.8404,C 0.2126,E1 8.6874,E2 284.1079} C_DIS
LIN {X -136.8612,Y 31.2686,Z 171,A 168.8799,B 8.8402,C 0.2166,E1 8.6865,E2 282.7373} C_DIS
LIN {X -138.0885,Y 25.3113,Z 171,A 171.4614,B 8.8401,C 0.222,E1 8.6851,E2 280.1457} C_DIS
LIN {X -138.9028,Y 20.3726,Z 171,A 173.6137,B 8.84,C 0.2261,E1 8.6842,E2 277.9814} C_DIS
LIN {X -139.3481,Y 17.0608,Z 171,A 175.8183,B 8.8402,C 0.2159,E1 8.6835,E2 275.6694} C_DIS
LIN {X -140.0105,Y 10.2884,Z 171,A 177.7307,B 8.8397,C 0.2385,E1 8.683,E2 273.8716} C_DIS
LIN {X -140.3493,Y 3.3471,Z 171,A -179.7474,B 8.8393,C 0.2519,E1 8.6827,E2 271.3928} C_DIS
LIN {X -140.3625,Y -2.7054,Z 171,A -176.9615,B 8.8393,C 0.2539,E1 8.6827,E2 268.569} C_DIS
LIN {X -140.0265,Y -10.0694,Z 171,A -174.1,B 8.8389,C 0.2651,E1 8.6831,E2 265.7293} C_DIS
LIN {X -139.3612,Y -16.9504,Z 171,A -170.9681,B 8.8389,C 0.2681,E1 8.684,E2 262.5602} C_DIS
LIN {X -138.7969,Y -21.0793,Z 171,A -169.1645,B 8.8387,C 0.2712,E1 8.6847,E2 260.7449} C_DIS
LIN {X -138.1922,Y -24.7318,Z 171,A -167.749,B 8.8386,C 0.2771,E1 8.6854,E2 259.3429} C_DIS
LIN {X -137.6264,Y -27.7091,Z 171,A -166.3869,B 8.8386,C 0.2785,E1 8.6861,E2 257.9657} C_DIS
LIN {X -136.8339,Y -31.3884,Z 171,A -164.9171,B 8.8383,C 0.2839,E1 8.687,E2 256.5057} C_DIS
LIN {X -136.0785,Y -34.5159,Z 171,A -163.5845,B 8.8383,C 0.2873,E1 8.6879,E2 255.1716} C_DIS
LIN {X -135.2441,Y -37.6533,Z 171,A -162.2344,B 8.8381,C 0.2905,E1 8.6889,E2 253.8193} C_DIS
LIN {X -134.3672,Y -40.6737,Z 171,A -160.8702,B 8.8381,C 0.2927,E1 8.69,E2 252.4456} C_DIS
LIN {X -133.1844,Y -44.3916,Z 171,A -159.285,B 8.8379,C 0.2971,E1 8.6914,E2 250.8625} C_DIS
LIN {X -131.7616,Y -48.4584,Z 171,A -157.4214,B 8.8379,C 0.3001,E1 8.6931,E2 248.9867} C_DIS
LIN {X -130.34,Y -52.1563,Z 171,A -155.7278,B 8.8377,C 0.3031,E1 8.6949,E2 247.2841} C_DIS
LIN {X -128.6749,Y -56.1394,Z 171,A -153.9377,B 8.8376,C 0.3073,E1 8.6968,E2 245.4916} C_DIS
LIN {X -126.8575,Y -60.1333,Z 171,A -152.2188,B 8.8374,C 0.3131,E1 8.6988,E2 243.7832} C_DIS
LIN {X -125.203,Y -63.5051,Z 171,A -150.7087,B 8.8372,C 0.3174,E1 8.7007,E2 242.277} C_DIS
LIN {X -123.3902,Y -66.9638,Z 171,A -148.9882,B 8.8372,C 0.3193,E1 8.703,E2 240.541} C_DIS
LIN {X -121.2593,Y -70.7501,Z 171,A -147.1378,B 8.837,C 0.3223,E1 8.7056,E2 238.6816} C_DIS
LIN {X -118.8584,Y -74.7126,Z 171,A -145.2395,B 8.8369,C 0.3267,E1 8.7084,E2 236.7833} C_DIS
LIN {X -116.3501,Y -78.5614,Z 171,A -143.372,B 8.8367,C 0.3313,E1 8.7113,E2 234.9178} C_DIS
LIN {X -113.8414,Y -82.1549,Z 171,A -141.5153,B 8.8366,C 0.3342,E1 8.7143,E2 233.0531} C_DIS
LIN {X -111.0348,Y -85.9098,Z 171,A -139.5987,B 8.8364,C 0.3385,E1 8.7175,E2 231.1369} C_DIS
LIN {X -108.1025,Y -89.5715,Z 171,A -137.6854,B 8.8363,C 0.3427,E1 8.7209,E2 229.2246} C_DIS
LIN {X -106.2857,Y -91.7201,Z 171,A -136.0977,B 8.8365,C 0.3373,E1 8.7239,E2 227.5797} C_DIS
LIN {X -103.3047,Y -95.065,Z 171,A -134.6848,B 8.836,C 0.3485,E1 8.7265,E2 226.2221} C_DIS
LIN {X -101.1694,Y -97.3353,Z 171,A -133.3305,B 8.836,C 0.3496,E1 8.7291,E2 224.8575} C_DIS
LIN {X -97.111,Y -101.3839,Z 171,A -131.013,B 8.8358,C 0.3546,E1 8.7337,E2 222.5437} C_DIS
LIN {X -93.8843,Y -104.3793,Z 171,A -129.1572,B 8.8358,C 0.3569,E1 8.7375,E2 220.6807} C_DIS
LIN {X -90.3754,Y -107.4315,Z 171,A -127.2627,B 8.8356,C 0.3604,E1 8.7416,E2 218.7871} C_DIS
LIN {X -86.8462,Y -110.304,Z 171,A -125.5872,B 8.8353,C 0.3669,E1 8.7452,E2 217.1358} C_DIS
LIN {X -79.4119,Y -115.7712,Z 171,A -121.6152,B 8.8353,C 0.3692,E1 8.7542,E2 213.1378} C_DIS
LIN {X -75.5548,Y -118.3246,Z 171,A -119.7348,B 8.8351,C 0.3722,E1 8.7586,E2 211.2586} C_DIS
LIN {X -71.8565,Y -120.6062,Z 171,A -117.9341,B 8.8351,C 0.3742,E1 8.7629,E2 209.4545} C_DIS
LIN {X -68.9582,Y -122.2867,Z 171,A -115.8234,B 8.8355,C 0.362,E1 8.7683,E2 207.2455} C_DIS
LIN {X -63.6913,Y -125.1082,Z 171,A -114.214,B 8.8347,C 0.3807,E1 8.772,E2 205.7459} C_DIS
LIN {X -60.7592,Y -126.5585,Z 171,A -112.8173,B 8.8347,C 0.381,E1 8.7755,E2 204.341} C_DIS
LIN {X -56.5642,Y -128.4906,Z 171,A -110.7989,B 8.8347,C 0.3806,E1 8.7807,E2 202.3051} C_DIS
LIN {X -52.7953,Y -130.0824,Z 171,A -109.2191,B 8.8346,C 0.3839,E1 8.7848,E2 200.737} C_DIS
LIN {X -49.488,Y -131.3761,Z 171,A -107.8347,B 8.8345,C 0.3865,E1 8.7883,E2 199.3609} C_DIS
LIN {X -46.608,Y -132.4266,Z 171,A -106.5303,B 8.8345,C 0.3865,E1 8.7918,E2 198.0494} C_DIS
LIN {X -43.0092,Y -133.6375,Z 171,A -104.9498,B 8.8345,C 0.3872,E1 8.796,E2 196.4645} C_DIS
LIN {X -39.6265,Y -134.6792,Z 171,A -103.6357,B 8.8343,C 0.3908,E1 8.7995,E2 195.1674} C_DIS
LIN {X -34.6065,Y -136.0555,Z 171,A -101.4077,B 8.8343,C 0.3901,E1 8.8055,E2 192.9253} C_DIS
LIN {X -31.4422,Y -136.8216,Z 171,A -100.0672,B 8.8343,C 0.3906,E1 8.8092,E2 191.5829} C_DIS
LIN {X -28.2563,Y -137.515,Z 171,A -98.683,B 8.8343,C 0.3902,E1 8.813,E2 190.1913} C_DIS
LIN {X -23.7902,Y -138.3591,Z 171,A -96.7727,B 8.8343,C 0.3899,E1 8.8182,E2 188.2732} C_DIS
LIN {X -20.533,Y -138.8799,Z 171,A -95.4244,B 8.8343,C 0.3903,E1 8.822,E2 186.9243} C_DIS
LIN {X -16.5771,Y -139.4058,Z 171,A -93.903,B 8.8343,C 0.3928,E1 8.8261,E2 185.4163} C_DIS
LIN {X -13.6252,Y -139.7254,Z 171,A -92.6118,B 8.8343,C 0.3914,E1 8.8298,E2 184.1143} C_DIS
LIN {X -9.3776,Y -140.0765,Z 171,A -90.927,B 8.8343,C 0.3927,E1 8.8344,E2 182.436} C_DIS
LIN {X -5.6397,Y -140.2748,Z 171,A -89.4168,B 8.8342,C 0.393,E1 8.8386,E2 180.9275} C_DIS
LIN {X -2.0401,Y -140.3736,Z 171,A -87.8494,B 8.8342,C 0.391,E1 8.8431,E2 179.3464} C_DIS
LIN {X 1.0238,Y -140.3815,Z 171,A -86.8823,B 8.834,C 0.3966,E1 8.8457,E2 178.416} C_DIS
Enddeposition()
LIN {X 1.0238,Y -140.3815,Z 171,A -86.8823,B 8.834,C 0.3966,E1 8.8457,E2 178.416} C_DIS
Startdeposition()
$VEL.CP = VEL_PRINT
LIN {X 0.0013,Y -141.3005,Z 171,A -87.7065,B 8.8336,C 0.4102,E1 8.8433,E2 179.3285} C_DIS
LIN {X -3.4614,Y -141.2568,Z 171,A -89.1007,B 8.8336,C 0.41,E1 8.8394,E2 180.722} C_DIS
LIN {X -7.7105,Y -141.0892,Z 171,A -90.8353,B 8.8336,C 0.4102,E1 8.8345,E2 182.4587} C_DIS
LIN {X -10.7292,Y -140.8911,Z 171,A -92.1082,B 8.8336,C 0.4111,E1 8.831,E2 183.7382} C_DIS
LIN {X -14.6289,Y -140.5398,Z 171,A -93.6392,B 8.8336,C 0.4097,E1 8.8267,E2 185.2623} C_DIS
LIN {X -18.2329,Y -140.117,Z 171,A -95.1048,B 8.8336,C 0.4092,E1 8.8227,E2 186.7276} C_DIS
LIN {X -21.6698,Y -139.6267,Z 171,A -96.512,B 8.8336,C 0.4088,E1 8.8188,E2 188.1352} C_DIS
LIN {X -25.0852,Y -139.0537,Z 171,A -97.919,B 8.8336,C 0.4083,E1 8.8149,E2 189.543} C_DIS
LIN {X -28.3332,Y -138.4284,Z 171,A -99.2631,B 8.8337,C 0.4078,E1 8.8112,E2 190.8879} C_DIS
LIN {X -31.7143,Y -137.6932,Z 171,A -100.6702,B 8.8337,C 0.4071,E1 8.8074,E2 192.2958} C_DIS
LIN {X -35.0778,Y -136.8751,Z 171,A -102.1366,B 8.8337,C 0.4075,E1 8.8034,E2 193.7709} C_DIS
LIN {X -39.3224,Y -135.7167,Z 171,A -103.8826,B 8.8337,C 0.4056,E1 8.7987,E2 195.5122} C_DIS
LIN {X -43.4227,Y -134.4611,Z 171,A -105.6182,B 8.8339,C 0.4042,E1 8.7941,E2 197.2477} C_DIS
LIN {X -46.8631,Y -133.3017,Z 171,A -107.0989,B 8.8339,C 0.4032,E1 8.7902,E2 198.7297} C_DIS
LIN {X -50.1187,Y -132.112,Z 171,A -108.5128,B 8.8339,C 0.4021,E1 8.7865,E2 200.1449} C_DIS
LIN {X -53.1904,Y -130.9046,Z 171,A -109.8744,B 8.8339,C 0.4012,E1 8.7829,E2 201.5096} C_DIS
LIN {X -56.388,Y -129.5592,Z 171,A -111.2827,B 8.8341,C 0.3998,E1 8.7793,E2 202.9182} C_DIS
LIN {X -59.6311,Y -128.099,Z 171,A -112.7251,B 8.8341,C 0.3982,E1 8.7757,E2 204.3607} C_DIS
LIN {X -62.7393,Y -126.6054,Z 171,A -114.1838,B 8.8341,C 0.3977,E1 8.772,E2 205.8273} C_DIS
LIN {X -66.2377,Y -124.8119,Z 171,A -115.7144,B 8.8343,C 0.3946,E1 8.7682,E2 207.3496} C_DIS
LIN {X -69.6182,Y -122.9599,Z 171,A -117.4183,B 8.8343,C 0.3951,E1 8.764,E2 209.0719} C_DIS
LIN {X -73.385,Y -120.7493,Z 171,A -119.1694,B 8.8343,C 0.3923,E1 8.7598,E2 210.8203} C_DIS
LIN {X -77.0498,Y -118.444,Z 171,A -120.9232,B 8.8345,C 0.3897,E1 8.7557,E2 212.5737} C_DIS
LIN {X -80.6287,Y -116.0373,Z 171,A -122.6974,B 8.8346,C 0.3875,E1 8.7516,E2 214.3509} C_DIS
LIN {X -84.1277,Y -113.5265,Z 171,A -124.4737,B 8.8347,C 0.3852,E1 8.7476,E2 216.1309} C_DIS
LIN {X -87.6131,Y -110.8592,Z 171,A -126.2747,B 8.8348,C 0.3826,E1 8.7436,E2 217.9344} C_DIS
LIN {X -90.9691,Y -108.1216,Z 171,A -128.0253,B 8.835,C 0.3794,E1 8.7398,E2 219.6837} C_DIS
LIN {X -94.1016,Y -105.4067,Z 171,A -129.7813,B 8.835,C 0.3777,E1 8.7361,E2 221.4491} C_DIS
LIN {X -97.4325,Y -102.3358,Z 171,A -131.6016,B 8.8352,C 0.3739,E1 8.7324,E2 223.2666} C_DIS
LIN {X -100.5296,Y -99.2956,Z 171,A -133.4317,B 8.8352,C 0.3716,E1 8.7288,E2 225.1054} C_DIS
LIN {X -103.7837,Y -95.8891,Z 171,A -135.3302,B 8.8355,C 0.3675,E1 8.7252,E2 227.0016} C_DIS
LIN {X -106.7227,Y -92.607,Z 171,A -137.1597,B 8.8355,C 0.3645,E1 8.7218,E2 228.8361} C_DIS
LIN {X -109.7336,Y -89.0187,Z 171,A -139.0646,B 8.8357,C 0.3605,E1 8.7184,E2 230.7408} C_DIS
LIN {X -112.4544,Y -85.5557,Z 171,A -140.8705,B 8.8359,C 0.3569,E1 8.7153,E2 232.5485} C_DIS
LIN {X -115.0231,Y -82.0691,Z 171,A -142.6319,B 8.836,C 0.353,E1 8.7124,E2 234.3098} C_DIS
LIN {X -117.484,Y -78.5058,Z 171,A -144.4131,B 8.8362,C 0.3493,E1 8.7096,E2 236.0934} C_DIS
LIN {X -119.9654,Y -74.6589,Z 171,A -146.3248,B 8.8363,C 0.3458,E1 8.7067,E2 238.0112} C_DIS
LIN {X -122.2776,Y -70.8084,Z 171,A -148.1388,B 8.8365,C 0.3412,E1 8.7042,E2 239.8232} C_DIS
LIN {X -124.3888,Y -67.0306,Z 171,A -149.9439,B 8.8366,C 0.3377,E1 8.7017,E2 241.6338} C_DIS
LIN {X -126.2119,Y -63.5299,Z 171,A -151.4761,B 8.8368,C 0.3325,E1 8.6998,E2 243.1562} C_DIS
LIN {X -127.7312,Y -60.4163,Z 171,A -152.9004,B 8.837,C 0.3292,E1 8.6981,E2 244.582} C_DIS
LIN {X -129.1737,Y -57.2665,Z 171,A -154.3261,B 8.837,C 0.3259,E1 8.6964,E2 246.0096} C_DIS
LIN {X -130.5481,Y -54.0599,Z 171,A -155.8887,B 8.8371,C 0.3246,E1 8.6947,E2 247.5903} C_DIS
LIN {X -132.0982,Y -50.1556,Z 171,A -157.498,B 8.8373,C 0.3185,E1 8.6931,E2 249.1863} C_DIS
LIN {X -133.2994,Y -46.8695,Z 171,A -158.9792,B 8.8374,C 0.3157,E1 8.6917,E2 250.6745} C_DIS
LIN {X -134.4617,Y -43.4207,Z 171,A -160.4297,B 8.8376,C 0.3113,E1 8.6904,E2 252.1207} C_DIS
LIN {X -135.4859,Y -40.1109,Z 171,A -162.0023,B 8.8376,C 0.3102,E1 8.6891,E2 253.7137} C_DIS
LIN {X -136.8127,Y -35.3237,Z 171,A -163.9707,B 8.8379,C 0.3039,E1 8.6877,E2 255.6747} C_DIS
LIN {X -137.6912,Y -31.7229,Z 171,A -165.4337,B 8.838,C 0.299,E1 8.6868,E2 257.1314} C_DIS
LIN {X -138.4277,Y -28.3366,Z 171,A -166.8246,B 8.8382,C 0.2948,E1 8.686,E2 258.5193} C_DIS
LIN {X -139.052,Y -25.0949,Z 171,A -168.2252,B 8.8382,C 0.292,E1 8.6853,E2 259.9267} C_DIS
LIN {X -139.6268,Y -21.6689,Z 171,A -169.6536,B 8.8384,C 0.2884,E1 8.6846,E2 261.3565} C_DIS
LIN {X -140.1164,Y -18.2376,Z 171,A -171.0608,B 8.8384,C 0.2844,E1 8.6841,E2 262.7627} C_DIS
LIN {X -140.506,Y -14.9431,Z 171,A -172.4552,B 8.8386,C 0.2813,E1 8.6837,E2 264.1622} C_DIS
LIN {X -140.8393,Y -11.3912,Z 171,A -173.9095,B 8.8387,C 0.2773,E1 8.6833,E2 265.6163} C_DIS
LIN {X -141.0883,Y -7.7283,Z 171,A -175.4506,B 8.8388,C 0.2739,E1 8.683,E2 267.1627} C_DIS
LIN {X -141.234,Y -4.2802,Z 171,A -176.8665,B 8.8389,C 0.2701,E1 8.6829,E2 268.5795} C_DIS
LIN {X -141.3008,Y -0.2868,Z 171,A -178.5789,B 8.839,C 0.2669,E1 8.6829,E2 270.3023} C_DIS
LIN {X -141.2566,Y 3.4654,Z 171,A 179.9361,B 8.8392,C 0.2619,E1 8.6829,E2 271.7812} C_DIS
LIN {X -141.0897,Y 7.7006,Z 171,A 178.1785,B 8.8393,C 0.2576,E1 8.6831,E2 273.5421} C_DIS
LIN {X -140.8439,Y 11.3366,Z 171,A 176.7333,B 8.8394,C 0.2527,E1 8.6834,E2 274.9818} C_DIS
LIN {X -140.5418,Y 14.6102,Z 171,A 175.3307,B 8.8395,C 0.25,E1 8.6838,E2 276.3919} C_DIS
LIN {X -140.1178,Y 18.2264,Z 171,A 173.8405,B 8.8396,C 0.246,E1 8.6843,E2 277.8824} C_DIS
LIN {X -139.6352,Y 21.6146,Z 171,A 172.4287,B 8.8397,C 0.2424,E1 8.6849,E2 279.296} C_DIS
LIN {X -139.0659,Y 25.0171,Z 171,A 171.006,B 8.8398,C 0.2388,E1 8.6856,E2 280.7203} C_DIS
LIN {X -138.4435,Y 28.2588,Z 171,A 169.5977,B 8.8399,C 0.2361,E1 8.6863,E2 282.1362} C_DIS
LIN {X -137.476,Y 32.6452,Z 171,A 167.8469,B 8.8401,C 0.2298,E1 8.6874,E2 283.8761} C_DIS
LIN {X -136.63,Y 36.0214,Z 171,A 166.3546,B 8.8401,C 0.2271,E1 8.6885,E2 285.3773} C_DIS
LIN {X -135.7061,Y 39.3588,Z 171,A 164.7903,B 8.8401,C 0.2259,E1 8.6897,E2 286.9606} C_DIS
LIN {X -134.4623,Y 43.419,Z 171,A 163.1793,B 8.8403,C 0.2192,E1 8.691,E2 288.5557} C_DIS
LIN {X -133.3031,Y 46.8589,Z 171,A 161.6821,B 8.8404,C 0.2156,E1 8.6924,E2 290.0546} C_DIS
LIN {X -132.1139,Y 50.1135,Z 171,A 160.2534,B 8.8405,C 0.2121,E1 8.6938,E2 291.4849} C_DIS
LIN {X -130.9073,Y 53.1839,Z 171,A 158.8793,B 8.8405,C 0.2091,E1 8.6952,E2 292.8622} C_DIS
LIN {X -129.5541,Y 56.3998,Z 171,A 157.4474,B 8.8407,C 0.2056,E1 8.6968,E2 294.2948} C_DIS
LIN {X -128.0958,Y 59.6379,Z 171,A 155.9939,B 8.8407,C 0.202,E1 8.6985,E2 295.7485} C_DIS
LIN {X -126.596,Y 62.7582,Z 171,A 154.5193,B 8.8407,C 0.1995,E1 8.7003,E2 297.2307} C_DIS
LIN {X -124.6167,Y 66.6065,Z 171,A 152.6968,B 8.8409,C 0.1961,E1 8.7026,E2 299.06} C_DIS
LIN {X -122.5178,Y 70.3933,Z 171,A 150.9209,B 8.8409,C 0.192,E1 8.7051,E2 300.8368} C_DIS
LIN {X -120.3056,Y 74.1098,Z 171,A 149.1613,B 8.8411,C 0.1877,E1 8.7076,E2 302.5952} C_DIS
LIN {X -117.9666,Y 77.7788,Z 171,A 147.3799,B 8.8411,C 0.1836,E1 8.7103,E2 304.377} C_DIS
LIN {X -115.5231,Y 81.3638,Z 171,A 145.5862,B 8.8412,C 0.18,E1 8.7132,E2 306.1732} C_DIS
LIN {X -112.977,Y 84.8642,Z 171,A 143.7954,B 8.8412,C 0.1765,E1 8.7162,E2 307.9668} C_DIS
LIN {X -110.3243,Y 88.2854,Z 171,A 142.0051,B 8.8414,C 0.173,E1 8.7192,E2 309.7597} C_DIS
LIN {X -107.6772,Y 91.4946,Z 171,A 140.2888,B 8.8414,C 0.1697,E1 8.7223,E2 311.478} C_DIS
LIN {X -104.6313,Y 94.9627,Z 171,A 138.404,B 8.8414,C 0.1659,E1 8.7258,E2 313.3626} C_DIS
LIN {X -101.4501,Y 98.3541,Z 171,A 136.5168,B 8.8416,C 0.1619,E1 8.7295,E2 315.2481} C_DIS
LIN {X -98.4165,Y 101.3897,Z 171,A 134.7368,B 8.8416,C 0.159,E1 8.733,E2 317.0315} C_DIS
LIN {X -95.2709,Y 104.3517,Z 171,A 132.9494,B 8.8416,C 0.1561,E1 8.7367,E2 318.8217} C_DIS
LIN {X -92.0332,Y 107.2174,Z 171,A 131.1825,B 8.8417,C 0.153,E1 8.7404,E2 320.5886} C_DIS
LIN {X -88.6286,Y 110.0482,Z 171,A 129.4044,B 8.8417,C 0.1493,E1 8.7442,E2 322.3629} C_DIS
LIN {X -85.236,Y 112.6964,Z 171,A 127.6274,B 8.8418,C 0.1467,E1 8.7482,E2 324.1423} C_DIS
LIN {X -81.7386,Y 115.2587,Z 171,A 125.8276,B 8.8418,C 0.1445,E1 8.7523,E2 325.9458} C_DIS
LIN {X -78.1079,Y 117.7496,Z 171,A 124.033,B 8.8419,C 0.1417,E1 8.7564,E2 327.7399} C_DIS
LIN {X -74.5272,Y 120.0473,Z 171,A 122.3003,B 8.8419,C 0.1391,E1 8.7605,E2 329.472} C_DIS
LIN {X -70.8186,Y 122.2717,Z 171,A 120.5345,B 8.8419,C 0.1367,E1 8.7647,E2 331.2378} C_DIS
LIN {X -67.0274,Y 124.3905,Z 171,A 118.736,B 8.842,C 0.1349,E1 8.7692,E2 333.0396} C_DIS
LIN {X -63.6357,Y 126.158,Z 171,A 117.2563,B 8.842,C 0.1315,E1 8.7728,E2 334.509} C_DIS
LIN {X -60.4221,Y 127.7284,Z 171,A 115.8022,B 8.842,C 0.1297,E1 8.7765,E2 335.9624} C_DIS
LIN {X -57.6105,Y 129.0198,Z 171,A 114.4559,B 8.842,C 0.1298,E1 8.7799,E2 337.3192} C_DIS
LIN {X -53.2051,Y 130.8987,Z 171,A 112.6422,B 8.8422,C 0.1253,E1 8.7845,E2 339.1153} C_DIS
LIN {X -50.1373,Y 132.105,Z 171,A 111.2473,B 8.8422,C 0.1249,E1 8.7882,E2 340.5165} C_DIS
LIN {X -46.8855,Y 133.2939,Z 171,A 109.7872,B 8.8422,C 0.1246,E1 8.792,E2 341.9826} C_DIS
LIN {X -43.4209,Y 134.4617,Z 171,A 108.3419,B 8.8422,C 0.1225,E1 8.7959,E2 343.4222} C_DIS
LIN {X -40.1102,Y 135.4861,Z 171,A 106.9285,B 8.8422,C 0.1214,E1 8.7996,E2 344.8356} C_DIS
LIN {X -36.7753,Y 136.4289,Z 171,A 105.3799,B 8.8422,C 0.123,E1 8.8039,E2 346.4013} C_DIS
LIN {X -32.2789,Y 137.5642,Z 171,A 103.4903,B 8.8422,C 0.1218,E1 8.809,E2 348.2908} C_DIS
LIN {X -28.4269,Y 138.4093,Z 171,A 101.9081,B 8.8422,C 0.1205,E1 8.8133,E2 349.8699} C_DIS
LIN {X -24.2868,Y 139.1966,Z 171,A 100.3198,B 8.8422,C 0.1173,E1 8.8176,E2 351.442} C_DIS
LIN {X -20.8318,Y 139.7564,Z 171,A 98.8506,B 8.8422,C 0.1176,E1 8.8217,E2 352.9167} C_DIS
LIN {X -17.3004,Y 140.2363,Z 171,A 97.34,B 8.8422,C 0.1183,E1 8.8259,E2 354.4346} C_DIS
LIN {X -12.9121,Y 140.7083,Z 171,A 95.6699,B 8.8422,C 0.1155,E1 8.8305,E2 356.0887} C_DIS
LIN {X -9.6141,Y 140.9725,Z 171,A 94.2679,B 8.8422,C 0.1163,E1 8.8344,E2 357.4976} C_DIS
LIN {X -5.9911,Y 141.1721,Z 171,A 92.8155,B 8.8422,C 0.1157,E1 8.8385,E2 358.9469} C_DIS
LIN {X -1.738,Y 141.289,Z 171,A 91.1353,B 8.8422,C 0.1147,E1 8.8431,E2 360.6206} C_DIS
LIN {X 1.7247,Y 141.2893,Z 171,A 89.6829,B 8.8422,C 0.1156,E1 8.8472,E2 362.0784} C_DIS
LIN {X 5.1845,Y 141.2036,Z 171,A 88.1732,B 8.8422,C 0.1178,E1 8.8515,E2 363.6009} C_DIS
LIN {X 9.6125,Y 140.9726,Z 171,A 86.4841,B 8.8422,C 0.1159,E1 8.8561,E2 365.2757} C_DIS
LIN {X 13.2991,Y 140.6712,Z 171,A 84.9164,B 8.8422,C 0.1176,E1 8.8605,E2 366.8513} C_DIS
LIN {X 17.2846,Y 140.2382,Z 171,A 83.3905,B 8.8422,C 0.1162,E1 8.8647,E2 368.3641} C_DIS
LIN {X 20.7265,Y 139.7718,Z 171,A 81.9849,B 8.8422,C 0.1167,E1 8.8686,E2 369.7689} C_DIS
LIN {X 24.158,Y 139.2197,Z 171,A 80.6116,B 8.8422,C 0.1166,E1 8.8724,E2 371.1373} C_DIS
LIN {X 27.555,Y 138.5867,Z 171,A 79.166,B 8.8422,C 0.1182,E1 8.8763,E2 372.588} C_DIS
LIN {X 30.9355,Y 137.8711,Z 171,A 77.6254,B 8.8422,C 0.1218,E1 8.8806,E2 374.1459} C_DIS
LIN {X 35.0689,Y 136.8774,Z 171,A 76.0294,B 8.8422,C 0.1204,E1 8.8849,E2 375.7253} C_DIS
LIN {X 39.3589,Y 135.706,Z 171,A 74.261,B 8.8422,C 0.1211,E1 8.8896,E2 377.489} C_DIS
LIN {X 42.6745,Y 134.7001,Z 171,A 72.8637,B 8.8422,C 0.1221,E1 8.8933,E2 378.8851} C_DIS
LIN {X 45.9642,Y 133.6133,Z 171,A 71.4015,B 8.8422,C 0.1246,E1 8.8972,E2 380.3544} C_DIS
LIN {X 50.1171,Y 132.1126,Z 171,A 69.6834,B 8.8422,C 0.1248,E1 8.9017,E2 382.0631} C_DIS
LIN {X 53.1919,Y 130.904,Z 171,A 68.3368,B 8.8422,C 0.1264,E1 8.9052,E2 383.4105} C_DIS
LIN {X 56.3933,Y 129.5569,Z 171,A 66.9598,B 8.8422,C 0.1273,E1 8.9087,E2 384.7834} C_DIS
LIN {X 59.6177,Y 128.1052,Z 171,A 65.5284,B 8.8421,C 0.1289,E1 8.9124,E2 386.2144} C_DIS
LIN {X 62.7304,Y 126.6097,Z 171,A 64.0868,B 8.8421,C 0.1316,E1 8.916,E2 387.6612} C_DIS
LIN {X 67.0024,Y 124.404,Z 171,A 62.1421,B 8.8421,C 0.1341,E1 8.9208,E2 389.6055} C_DIS
LIN {X 70.8104,Y 122.2764,Z 171,A 60.3912,B 8.842,C 0.1362,E1 8.925,E2 391.3542} C_DIS
LIN {X 74.5338,Y 120.0432,Z 171,A 58.6637,B 8.842,C 0.1381,E1 8.9291,E2 393.0776} C_DIS
LIN {X 78.0995,Y 117.7552,Z 171,A 56.9054,B 8.842,C 0.1416,E1 8.9333,E2 394.8414} C_DIS
LIN {X 81.6626,Y 115.3123,Z 171,A 55.1836,B 8.8419,C 0.1438,E1 8.9372,E2 396.5596} C_DIS
LIN {X 85.1792,Y 112.7393,Z 171,A 53.4484,B 8.8419,C 0.1462,E1 8.9411,E2 398.2911} C_DIS
LIN {X 88.5952,Y 110.0752,Z 171,A 51.6972,B 8.8418,C 0.1492,E1 8.9449,E2 400.0419} C_DIS
LIN {X 91.9909,Y 107.2539,Z 171,A 49.9263,B 8.8418,C 0.1521,E1 8.9487,E2 401.8108} C_DIS
LIN {X 95.2498,Y 104.3708,Z 171,A 48.1824,B 8.8417,C 0.155,E1 8.9523,E2 403.5526} C_DIS
LIN {X 98.3506,Y 101.4534,Z 171,A 46.4889,B 8.8417,C 0.1577,E1 8.9557,E2 405.2425} C_DIS
LIN {X 101.403,Y 98.4028,Z 171,A 44.743,B 8.8416,C 0.1612,E1 8.9592,E2 406.9884} C_DIS
LIN {X 104.3699,Y 95.2509,Z 171,A 42.9945,B 8.8416,C 0.1647,E1 8.9625,E2 408.7367} C_DIS
LIN {X 107.2535,Y 91.9914,Z 171,A 41.2616,B 8.8415,C 0.1678,E1 8.9657,E2 410.4663} C_DIS
LIN {X 110.0748,Y 88.5957,Z 171,A 39.5256,B 8.8414,C 0.1706,E1 8.9687,E2 412.1961} C_DIS
LIN {X 112.6885,Y 85.2465,Z 171,A 37.7975,B 8.8414,C 0.1747,E1 8.9717,E2 413.9257} C_DIS
LIN {X 115.2972,Y 81.684,Z 171,A 36.0364,B 8.8413,C 0.1782,E1 8.9745,E2 415.6838} C_DIS
LIN {X 117.7537,Y 78.1017,Z 171,A 34.3319,B 8.8412,C 0.1811,E1 8.9772,E2 417.3819} C_DIS
LIN {X 120.0402,Y 74.5387,Z 171,A 32.6095,B 8.8412,C 0.1854,E1 8.9798,E2 419.1061} C_DIS
LIN {X 122.2618,Y 70.8357,Z 171,A 30.8788,B 8.841,C 0.1893,E1 8.9822,E2 420.835} C_DIS
LIN {X 124.3913,Y 67.026,Z 171,A 29.1173,B 8.841,C 0.1936,E1 8.9846,E2 422.5966} C_DIS
LIN {X 126.2111,Y 63.5313,Z 171,A 27.6309,B 8.8409,C 0.1951,E1 8.9865,E2 424.0697} C_DIS
LIN {X 127.7372,Y 60.4037,Z 171,A 26.2488,B 8.8409,C 0.1981,E1 8.9881,E2 425.4489} C_DIS
LIN {X 129.174,Y 57.2659,Z 171,A 24.8656,B 8.8408,C 0.2014,E1 8.9897,E2 426.8308} C_DIS
LIN {X 130.5338,Y 54.0941,Z 171,A 23.4885,B 8.8407,C 0.2047,E1 8.9912,E2 428.2061} C_DIS
LIN {X 131.8295,Y 50.8549,Z 171,A 22.0732,B 8.8406,C 0.2085,E1 8.9926,E2 429.6225} C_DIS
LIN {X 133.3019,Y 46.8623,Z 171,A 20.3524,B 8.8405,C 0.213,E1 8.9943,E2 431.3439} C_DIS
LIN {X 134.4614,Y 43.4217,Z 171,A 18.8043,B 8.8403,C 0.2188,E1 8.9956,E2 432.9027} C_DIS
LIN {X 135.7697,Y 39.1417,Z 171,A 17.0182,B 8.8403,C 0.2232,E1 8.9971,E2 434.6866} C_DIS
LIN {X 137.0645,Y 34.3315,Z 171,A 15.1747,B 8.8402,C 0.2248,E1 8.9983,E2 436.5088} C_DIS
LIN {X 137.8703,Y 30.9389,Z 171,A 13.788,B 8.8402,C 0.2281,E1 8.9992,E2 437.8932} C_DIS
LIN {X 138.5857,Y 27.5603,Z 171,A 12.4124,B 8.84,C 0.2315,E1 9,E2 439.2668} C_DIS
LIN {X 139.2185,Y 24.1643,Z 171,A 11.0373,B 8.84,C 0.2349,E1 9.0007,E2 440.6398} C_DIS
LIN {X 139.7682,Y 20.7514,Z 171,A 9.6804,B 8.8399,C 0.2379,E1 9.0012,E2 441.992} C_DIS
LIN {X 140.2362,Y 17.3007,Z 171,A 8.2479,B 8.8397,C 0.2424,E1 9.0018,E2 443.4283} C_DIS
LIN {X 140.6187,Y 13.846,Z 171,A 6.8652,B 8.8397,C 0.2459,E1 9.0022,E2 444.8088} C_DIS
LIN {X 140.9469,Y 9.9643,Z 171,A 5.2496,B 8.8395,C 0.2513,E1 9.0025,E2 446.4304} C_DIS
LIN {X 141.1721,Y 5.9909,Z 171,A 3.7179,B 8.8395,C 0.254,E1 9.0027,E2 447.9529} C_DIS
LIN {X 141.2759,Y 2.5293,Z 171,A 2.3125,B 8.8393,C 0.2581,E1 9.0028,E2 449.3598} C_DIS
LIN {X 141.2891,Y -1.7346,Z 171,A 0.6305,B 8.8392,C 0.2621,E1 9.0028,E2 451.0373} C_DIS
LIN {X 141.2032,Y -5.1955,Z 171,A -0.74,B 8.8391,C 0.2654,E1 9.0027,E2 452.4048} C_DIS
LIN {X 141.0323,Y -8.6662,Z 171,A -2.1182,B 8.839,C 0.2688,E1 9.0025,E2 453.7803} C_DIS
LIN {X 140.7321,Y -12.6596,Z 171,A -3.7928,B 8.8388,C 0.2746,E1 9.0021,E2 455.4632} C_DIS
LIN {X 140.3491,Y -16.3544,Z 171,A -5.2395,B 8.8388,C 0.2776,E1 9.0017,E2 456.9035} C_DIS
LIN {X 139.8825,Y -19.9518,Z 171,A -6.645,B 8.8386,C 0.2803,E1 9.0011,E2 458.3019} C_DIS
LIN {X 139.3515,Y -23.374,Z 171,A -8.0244,B 8.8386,C 0.2838,E1 9.0005,E2 459.6795} C_DIS
LIN {X 138.7368,Y -26.7831,Z 171,A -9.4603,B 8.8384,C 0.2886,E1 8.9998,E2 461.1208} C_DIS
LIN {X 137.9844,Y -30.428,Z 171,A -10.9974,B 8.8382,C 0.2935,E1 8.9989,E2 462.6631} C_DIS
LIN {X 137.0724,Y -34.3004,Z 171,A -12.4808,B 8.8382,C 0.2951,E1 8.9979,E2 464.1312} C_DIS
LIN {X 136.1946,Y -37.6344,Z 171,A -13.8566,B 8.838,C 0.2986,E1 8.9969,E2 465.5056} C_DIS
LIN {X 134.9973,Y -41.7253,Z 171,A -15.5609,B 8.8379,C 0.3028,E1 8.9955,E2 467.2085} C_DIS
LIN {X 133.9195,Y -45.0653,Z 171,A -16.9712,B 8.8378,C 0.3065,E1 8.9943,E2 468.6186} C_DIS
LIN {X 132.7295,Y -48.4592,Z 171,A -18.3977,B 8.8376,C 0.3098,E1 8.993,E2 470.0425} C_DIS
LIN {X 131.2753,Y -52.271,Z 171,A -20.13,B 8.8374,C 0.3161,E1 8.9912,E2 471.7866} C_DIS
LIN {X 129.5601,Y -56.386,Z 171,A -21.8129,B 8.8374,C 0.3182,E1 8.9894,E2 473.4551} C_DIS
LIN {X 128.1076,Y -59.6124,Z 171,A -23.2527,B 8.8372,C 0.3221,E1 8.9877,E2 474.897} C_DIS
LIN {X 126.532,Y -62.8881,Z 171,A -24.7136,B 8.8371,C 0.3257,E1 8.9859,E2 476.3577} C_DIS
LIN {X 124.3915,Y -67.0257,Z 171,A -26.5887,B 8.8369,C 0.3303,E1 8.9835,E2 478.2331} C_DIS
LIN {X 122.2753,Y -70.8124,Z 171,A -28.3205,B 8.8368,C 0.3342,E1 8.9811,E2 479.9631} C_DIS
LIN {X 120.0486,Y -74.5251,Z 171,A -30.0641,B 8.8366,C 0.3384,E1 8.9786,E2 481.707} C_DIS
LIN {X 117.7507,Y -78.1062,Z 171,A -31.7872,B 8.8364,C 0.3427,E1 8.9759,E2 483.4316} C_DIS
LIN {X 115.3179,Y -81.6548,Z 171,A -33.4939,B 8.8364,C 0.346,E1 8.9732,E2 485.1351} C_DIS
LIN {X 112.7708,Y -85.1375,Z 171,A -35.2091,B 8.8362,C 0.3494,E1 8.9704,E2 486.8476} C_DIS
LIN {X 110.0716,Y -88.5996,Z 171,A -36.9758,B 8.836,C 0.3533,E1 8.9673,E2 488.6144} C_DIS
LIN {X 107.2538,Y -91.991,Z 171,A -38.7361,B 8.8359,C 0.3568,E1 8.9641,E2 490.3728} C_DIS
LIN {X 104.386,Y -95.2331,Z 171,A -40.4695,B 8.8358,C 0.3602,E1 8.9609,E2 492.1052} C_DIS
LIN {X 101.4043,Y -98.4013,Z 171,A -42.1902,B 8.8356,C 0.3631,E1 8.9576,E2 493.822} C_DIS
LIN {X 98.4018,Y -101.4038,Z 171,A -43.9191,B 8.8355,C 0.3669,E1 8.9541,E2 495.5534} C_DIS
LIN {X 95.2491,Y -104.3715,Z 171,A -45.6685,B 8.8353,C 0.3703,E1 8.9506,E2 497.3038} C_DIS
LIN {X 92.0067,Y -107.2403,Z 171,A -47.396,B 8.8353,C 0.3732,E1 8.9469,E2 499.0293} C_DIS
LIN {X 88.6001,Y -110.0712,Z 171,A -49.139,B 8.8351,C 0.3755,E1 8.9432,E2 500.767} C_DIS
LIN {X 85.1879,Y -112.7327,Z 171,A -50.8864,B 8.835,C 0.3786,E1 8.9393,E2 502.5151} C_DIS
LIN {X 81.6943,Y -115.2899,Z 171,A -52.6349,B 8.8349,C 0.3815,E1 8.9353,E2 504.2643} C_DIS
LIN {X 78.108,Y -117.7495,Z 171,A -54.3837,B 8.8347,C 0.3843,E1 8.9313,E2 506.0128} C_DIS
LIN {X 74.546,Y -120.0356,Z 171,A -56.0771,B 8.8347,C 0.3866,E1 8.9273,E2 507.7047} C_DIS
LIN {X 70.8413,Y -122.2585,Z 171,A -57.8145,B 8.8345,C 0.389,E1 8.9231,E2 509.4418} C_DIS
LIN {X 67.0325,Y -124.3878,Z 171,A -59.5909,B 8.8345,C 0.3918,E1 8.9188,E2 511.2207} C_DIS
LIN {X 63.5317,Y -126.2109,Z 171,A -61.0894,B 8.8345,C 0.3918,E1 8.9151,E2 512.707} C_DIS
LIN {X 60.4147,Y -127.7319,Z 171,A -62.4812,B 8.8343,C 0.3935,E1 8.9116,E2 514.0981} C_DIS
LIN {X 57.6451,Y -129.0044,Z 171,A -63.7587,B 8.8343,C 0.396,E1 8.9083,E2 515.382} C_DIS
LIN {X 54.0725,Y -130.5428,Z 171,A -65.3919,B 8.8341,C 0.3992,E1 8.9041,E2 517.0238} C_DIS
LIN {X 50.1248,Y -132.1097,Z 171,A -66.9797,B 8.8341,C 0.3983,E1 8.9,E2 518.5953} C_DIS
LIN {X 46.6561,Y -133.3734,Z 171,A -68.5999,B 8.8339,C 0.4025,E1 8.8957,E2 520.2329} C_DIS
LIN {X 42.5108,Y -134.7524,Z 171,A -70.3745,B 8.8339,C 0.4044,E1 8.891,E2 522.0092} C_DIS
LIN {X 38.4438,Y -135.9683,Z 171,A -71.9496,B 8.8339,C 0.4029,E1 8.8868,E2 523.5662} C_DIS
LIN {X 34.3159,Y -137.0685,Z 171,A -73.6624,B 8.8339,C 0.4039,E1 8.8822,E2 525.2777} C_DIS
LIN {X 30.9547,Y -137.8667,Z 171,A -75.0552,B 8.8339,C 0.4049,E1 8.8784,E2 526.6704} C_DIS
LIN {X 27.1472,Y -138.6672,Z 171,A -76.7237,B 8.8337,C 0.4079,E1 8.8738,E2 528.3519} C_DIS
LIN {X 23.4003,Y -139.3471,Z 171,A -78.1722,B 8.8337,C 0.4068,E1 8.8698,E2 529.7887} C_DIS
LIN {X 19.9803,Y -139.8784,Z 171,A -79.5689,B 8.8337,C 0.4074,E1 8.866,E2 531.1853} C_DIS
LIN {X 16.3536,Y -140.3492,Z 171,A -81.0395,B 8.8337,C 0.4079,E1 8.8619,E2 532.6552} C_DIS
LIN {X 12.9073,Y -140.7088,Z 171,A -82.4274,B 8.8337,C 0.4081,E1 8.858,E2 534.0418} C_DIS
LIN {X 9.6171,Y -140.9723,Z 171,A -83.8207,B 8.8337,C 0.4097,E1 8.8541,E2 535.443} C_DIS
LIN {X 5.987,Y -141.1723,Z 171,A -85.4004,B 8.8335,C 0.4122,E1 8.8497,E2 537.0373} C_DIS
LIN {X 1.7333,Y -141.2891,Z 171,A -86.9602,B 8.8336,C 0.4092,E1 8.8454,E2 538.5762} C_DIS
LIN {X 1.7333,Y -141.2891,Z 171,A -86.9602,B 8.8336,C 0.4092,E1 8.8454,E2 538.5762} C_DIS
Enddeposition()
LIN {X 0.959,Y -132.3535,Z 172,A -87.4152,B 9.2703,C 0.3485,E1 9.2792,E2 538.5796} C_DIS
Startdeposition()
$VEL.CP = VEL_PRINT
LIN {X 3.2449,Y -132.3195,Z 172,A -86.0105,B 9.2706,C 0.3401,E1 9.2833,E2 537.1235} C_DIS
LIN {X 6.618,Y -132.1929,Z 172,A -84.66,B 9.2706,C 0.3419,E1 9.287,E2 535.7858} C_DIS
LIN {X 9.7347,Y -132,Z 172,A -83.298,B 9.2706,C 0.3413,E1 9.2908,E2 534.4219} C_DIS
LIN {X 13.407,Y -131.6798,Z 172,A -81.7396,B 9.2706,C 0.3413,E1 9.2952,E2 532.8672} C_DIS
LIN {X 16.3319,Y -131.3486,Z 172,A -80.4631,B 9.2706,C 0.3408,E1 9.2987,E2 531.5897} C_DIS
LIN {X 19.5444,Y -130.9093,Z 172,A -79.0484,B 9.2706,C 0.3398,E1 9.3026,E2 530.1727} C_DIS
LIN {X 22.7459,Y -130.3905,Z 172,A -77.6862,B 9.2706,C 0.3398,E1 9.3064,E2 528.8148} C_DIS
LIN {X 25.8242,Y -129.8159,Z 172,A -76.2925,B 9.2707,C 0.3381,E1 9.3102,E2 527.4155} C_DIS
LIN {X 29.0012,Y -129.1428,Z 172,A -74.8582,B 9.2707,C 0.3365,E1 9.3141,E2 525.9768} C_DIS
LIN {X 32.2852,Y -128.3606,Z 172,A -73.4414,B 9.2707,C 0.3362,E1 9.3179,E2 524.5644} C_DIS
LIN {X 35.4226,Y -127.5303,Z 172,A -72.0442,B 9.2708,C 0.3351,E1 9.3217,E2 523.1672} C_DIS
LIN {X 39.2114,Y -126.4175,Z 172,A -70.1926,B 9.271,C 0.3305,E1 9.3267,E2 521.2968} C_DIS
LIN {X 42.9583,Y -125.1936,Z 172,A -68.5601,B 9.271,C 0.3303,E1 9.331,E2 519.6722} C_DIS
LIN {X 46.2692,Y -124.0074,Z 172,A -67.1768,B 9.271,C 0.3315,E1 9.3346,E2 518.3048} C_DIS
LIN {X 49.1505,Y -122.8943,Z 172,A -65.746,B 9.271,C 0.3279,E1 9.3384,E2 516.8614} C_DIS
LIN {X 52.2681,Y -121.6008,Z 172,A -64.3583,B 9.271,C 0.3277,E1 9.3419,E2 515.4815} C_DIS
LIN {X 55.1131,Y -120.3388,Z 172,A -63.0224,B 9.2711,C 0.3262,E1 9.3453,E2 514.146} C_DIS
LIN {X 58.0459,Y -118.9522,Z 172,A -61.6225,B 9.2712,C 0.3243,E1 9.3488,E2 512.7454} C_DIS
LIN {X 61.0776,Y -117.4241,Z 172,A -60.2044,B 9.2712,C 0.3233,E1 9.3523,E2 511.3324} C_DIS
LIN {X 63.8067,Y -115.9655,Z 172,A -58.8456,B 9.2713,C 0.3209,E1 9.3557,E2 509.9702} C_DIS
LIN {X 66.6103,Y -114.3781,Z 172,A -57.4383,B 9.2714,C 0.3185,E1 9.3591,E2 508.56} C_DIS
LIN {X 69.4792,Y -112.6584,Z 172,A -55.9916,B 9.2714,C 0.3162,E1 9.3625,E2 507.1122} C_DIS
LIN {X 72.9212,Y -110.4613,Z 172,A -54.1256,B 9.2717,C 0.3111,E1 9.367,E2 505.2325} C_DIS
LIN {X 76.3332,Y -108.1315,Z 172,A -52.498,B 9.2717,C 0.3114,E1 9.3706,E2 503.623} C_DIS
LIN {X 78.8457,Y -106.3136,Z 172,A -51.0356,B 9.2718,C 0.3064,E1 9.374,E2 502.1445} C_DIS
LIN {X 82.0549,Y -103.8571,Z 172,A -49.282,B 9.2719,C 0.303,E1 9.3778,E2 500.3888} C_DIS
LIN {X 85.2666,Y -101.2365,Z 172,A -47.5142,B 9.272,C 0.3001,E1 9.3816,E2 498.6224} C_DIS
LIN {X 88.4833,Y -98.4374,Z 172,A -45.7202,B 9.272,C 0.2975,E1 9.3854,E2 496.8331} C_DIS
LIN {X 91.7982,Y -95.354,Z 172,A -43.7533,B 9.2722,C 0.2933,E1 9.3894,E2 494.8633} C_DIS
LIN {X 94.7793,Y -92.3916,Z 172,A -41.9483,B 9.2723,C 0.2897,E1 9.3929,E2 493.0583} C_DIS
LIN {X 98.0309,Y -88.9331,Z 172,A -40.0486,B 9.2723,C 0.2886,E1 9.3965,E2 491.1756} C_DIS
LIN {X 100.7178,Y -85.8786,Z 172,A -38.3278,B 9.2725,C 0.2855,E1 9.3996,E2 489.4579} C_DIS
LIN {X 102.8714,Y -83.2868,Z 172,A -36.7574,B 9.2727,C 0.2796,E1 9.4024,E2 487.8722} C_DIS
LIN {X 105.4741,Y -79.9653,Z 172,A -35.1261,B 9.2727,C 0.2796,E1 9.4052,E2 486.2631} C_DIS
LIN {X 107.2702,Y -77.539,Z 172,A -33.7958,B 9.2727,C 0.276,E1 9.4074,E2 484.9285} C_DIS
LIN {X 109.134,Y -74.8928,Z 172,A -32.3868,B 9.2729,C 0.2724,E1 9.4096,E2 483.5171} C_DIS
LIN {X 110.9521,Y -72.1721,Z 172,A -31.0203,B 9.2729,C 0.27,E1 9.4117,E2 482.1552} C_DIS
LIN {X 112.6874,Y -69.4318,Z 172,A -29.6046,B 9.273,C 0.2662,E1 9.4138,E2 480.7366} C_DIS
LIN {X 114.4413,Y -66.5012,Z 172,A -28.1825,B 9.2731,C 0.2636,E1 9.4158,E2 479.3199} C_DIS
LIN {X 115.9628,Y -63.8116,Z 172,A -26.8527,B 9.2732,C 0.2603,E1 9.4176,E2 477.9896} C_DIS
LIN {X 117.5476,Y -60.8423,Z 172,A -25.3267,B 9.2734,C 0.255,E1 9.4196,E2 476.4537} C_DIS
LIN {X 118.9984,Y -57.9522,Z 172,A -24.0342,B 9.2734,C 0.2537,E1 9.4212,E2 475.1728} C_DIS
LIN {X 120.3249,Y -55.143,Z 172,A -22.7123,B 9.2734,C 0.2506,E1 9.4227,E2 473.8522} C_DIS
LIN {X 121.6533,Y -52.1468,Z 172,A -21.3026,B 9.2736,C 0.2469,E1 9.4243,E2 472.4421} C_DIS
LIN {X 122.9446,Y -49.0257,Z 172,A -19.8748,B 9.2736,C 0.2437,E1 9.4258,E2 471.017} C_DIS
LIN {X 124.1103,Y -45.9945,Z 172,A -18.491,B 9.2737,C 0.2404,E1 9.4272,E2 469.6344} C_DIS
LIN {X 125.2004,Y -42.9386,Z 172,A -17.1121,B 9.2738,C 0.237,E1 9.4284,E2 468.2571} C_DIS
LIN {X 126.3557,Y -39.4133,Z 172,A -15.3231,B 9.274,C 0.2284,E1 9.43,E2 466.4441} C_DIS
LIN {X 127.5579,Y -35.324,Z 172,A -13.7136,B 9.274,C 0.2285,E1 9.4312,E2 464.8614} C_DIS
LIN {X 128.3804,Y -32.2072,Z 172,A -12.3302,B 9.2741,C 0.2248,E1 9.4322,E2 463.4781} C_DIS
LIN {X 129.1502,Y -28.9688,Z 172,A -10.918,B 9.2742,C 0.2214,E1 9.433,E2 462.0679} C_DIS
LIN {X 129.8427,Y -25.6921,Z 172,A -9.5027,B 9.2742,C 0.218,E1 9.4338,E2 460.6553} C_DIS
LIN {X 130.436,Y -22.4874,Z 172,A -8.1385,B 9.2744,C 0.215,E1 9.4345,E2 459.2955} C_DIS
LIN {X 130.9283,Y -19.4163,Z 172,A -6.7642,B 9.2744,C 0.2105,E1 9.4351,E2 457.9164} C_DIS
LIN {X 131.3641,Y -16.2017,Z 172,A -5.3844,B 9.2745,C 0.207,E1 9.4356,E2 456.5382} C_DIS
LIN {X 131.7214,Y -12.9745,Z 172,A -3.881,B 9.2747,C 0.2006,E1 9.436,E2 455.0214} C_DIS
LIN {X 132.1098,Y -8.1091,Z 172,A -1.9349,B 9.2747,C 0.1983,E1 9.4364,E2 453.0935} C_DIS
LIN {X 132.2745,Y -4.7352,Z 172,A -0.5194,B 9.2747,C 0.1951,E1 9.4366,E2 451.6823} C_DIS
LIN {X 132.3534,Y -1.3452,Z 172,A 0.8295,B 9.2748,C 0.1935,E1 9.4366,E2 450.3465} C_DIS
LIN {X 132.3477,Y 1.7512,Z 172,A 2.2484,B 9.2749,C 0.1878,E1 9.4366,E2 448.9168} C_DIS
LIN {X 132.2643,Y 4.9968,Z 172,A 3.6916,B 9.275,C 0.1829,E1 9.4365,E2 447.4677} C_DIS
LIN {X 132.101,Y 8.2525,Z 172,A 5.0803,B 9.2751,C 0.1793,E1 9.4363,E2 446.0803} C_DIS
LIN {X 131.8594,Y 11.4878,Z 172,A 6.4161,B 9.2751,C 0.1768,E1 9.4359,E2 444.7516} C_DIS
LIN {X 131.5387,Y 14.718,Z 172,A 7.7957,B 9.2752,C 0.1733,E1 9.4355,E2 443.3739} C_DIS
LIN {X 131.1396,Y 17.9357,Z 172,A 9.2028,B 9.2752,C 0.1692,E1 9.435,E2 441.9652} C_DIS
LIN {X 130.6791,Y 21.0303,Z 172,A 10.5788,B 9.2754,C 0.1649,E1 9.4344,E2 440.5853} C_DIS
LIN {X 130.1232,Y 24.2296,Z 172,A 11.9152,B 9.2754,C 0.1624,E1 9.4338,E2 439.2562} C_DIS
LIN {X 129.4895,Y 27.4126,Z 172,A 13.3101,B 9.2754,C 0.1586,E1 9.433,E2 437.8613} C_DIS
LIN {X 128.7453,Y 30.7157,Z 172,A 14.7369,B 9.2755,C 0.1554,E1 9.4321,E2 436.4379} C_DIS
LIN {X 127.9531,Y 33.8638,Z 172,A 16.1203,B 9.2755,C 0.1519,E1 9.4311,E2 435.0561} C_DIS
LIN {X 126.9744,Y 37.3658,Z 172,A 17.5623,B 9.2756,C 0.1505,E1 9.43,E2 433.6288} C_DIS
LIN {X 126.1345,Y 40.1097,Z 172,A 18.9718,B 9.2757,C 0.1433,E1 9.4288,E2 432.1982} C_DIS
LIN {X 125.1594,Y 43.0568,Z 172,A 20.2146,B 9.2757,C 0.1419,E1 9.4277,E2 430.9666} C_DIS
LIN {X 124.069,Y 46.1047,Z 172,A 21.594,B 9.2758,C 0.1386,E1 9.4264,E2 429.5887} C_DIS
LIN {X 122.761,Y 49.4811,Z 172,A 23.0888,B 9.2758,C 0.136,E1 9.4249,E2 428.1016} C_DIS
LIN {X 121.5991,Y 52.2722,Z 172,A 24.4293,B 9.2759,C 0.1318,E1 9.4234,E2 426.7564} C_DIS
LIN {X 120.3366,Y 55.1178,Z 172,A 25.7546,B 9.2759,C 0.1288,E1 9.4219,E2 425.4329} C_DIS
LIN {X 118.9483,Y 58.0538,Z 172,A 27.138,B 9.2759,C 0.1256,E1 9.4202,E2 424.0513} C_DIS
LIN {X 117.4291,Y 61.0681,Z 172,A 28.5563,B 9.276,C 0.1228,E1 9.4184,E2 422.6373} C_DIS
LIN {X 115.9532,Y 63.8288,Z 172,A 29.9167,B 9.276,C 0.1193,E1 9.4166,E2 421.2754} C_DIS
LIN {X 114.3555,Y 66.6494,Z 172,A 31.331,B 9.2761,C 0.1156,E1 9.4147,E2 419.859} C_DIS
LIN {X 112.6136,Y 69.5522,Z 172,A 32.758,B 9.2761,C 0.1128,E1 9.4126,E2 418.4358} C_DIS
LIN {X 110.9459,Y 72.1816,Z 172,A 34.1049,B 9.2761,C 0.1096,E1 9.4105,E2 417.0882} C_DIS
LIN {X 109.0682,Y 74.9887,Z 172,A 35.5305,B 9.2762,C 0.1069,E1 9.4083,E2 415.6662} C_DIS
LIN {X 107.188,Y 77.6523,Z 172,A 36.9028,B 9.2762,C 0.1044,E1 9.4061,E2 414.2979} C_DIS
LIN {X 104.8921,Y 80.7278,Z 172,A 38.5723,B 9.2762,C 0.1005,E1 9.4033,E2 412.6267} C_DIS
LIN {X 102.3408,Y 83.9379,Z 172,A 40.3238,B 9.2763,C 0.097,E1 9.4002,E2 410.8771} C_DIS
LIN {X 99.7353,Y 87.0174,Z 172,A 42.0633,B 9.2763,C 0.0933,E1 9.3971,E2 409.1378} C_DIS
LIN {X 96.9552,Y 90.1047,Z 172,A 43.9343,B 9.2764,C 0.088,E1 9.3935,E2 407.2574} C_DIS
LIN {X 94.1712,Y 93.0112,Z 172,A 45.5336,B 9.2764,C 0.0875,E1 9.3904,E2 405.6746} C_DIS
LIN {X 91.8075,Y 95.345,Z 172,A 47.1133,B 9.2764,C 0.0815,E1 9.3872,E2 404.0774} C_DIS
LIN {X 88.9009,Y 98.0602,Z 172,A 48.8087,B 9.2764,C 0.0788,E1 9.3837,E2 402.3847} C_DIS
LIN {X 85.8369,Y 100.7532,Z 172,A 50.4233,B 9.2764,C 0.0787,E1 9.3804,E2 400.7876} C_DIS
LIN {X 82.7101,Y 103.336,Z 172,A 52.2955,B 9.2765,C 0.073,E1 9.3763,E2 398.9011} C_DIS
LIN {X 79.5328,Y 105.8005,Z 172,A 54.0166,B 9.2765,C 0.0704,E1 9.3725,E2 397.1821} C_DIS
LIN {X 76.2263,Y 108.2068,Z 172,A 55.627,B 9.2765,C 0.0709,E1 9.3688,E2 395.5904} C_DIS
LIN {X 73.461,Y 110.1029,Z 172,A 57.0355,B 9.2765,C 0.0694,E1 9.3656,E2 394.1867} C_DIS
LIN {X 70.8109,Y 111.8258,Z 172,A 58.4198,B 9.2765,C 0.067,E1 9.3623,E2 392.8004} C_DIS
LIN {X 67.9285,Y 113.5998,Z 172,A 59.8727,B 9.2766,C 0.0651,E1 9.3589,E2 391.3488} C_DIS
Enddeposition()
END
